LIN {X 0,Y 238.062,Z 428.573,A -85,B 0,C 180,E1 -19850.136,E2 -19850.136} C_VEL
LIN {X 0,Y 238.193,Z 430.072,A -85,B 0,C 180,E1 -19851.55,E2 -19851.55} C_VEL
LIN {X 0,Y 238.018,Z 431.292,A -85,B 0,C 180,E1 -19852.418,E2 -19852.418} C_VEL
LIN {X 0,Y 236.97,Z 433.958,A -85,B 0,C 180,E1 -19853.62,E2 -19853.62} C_VEL
LIN {X 0,Y 235.097,Z 438.66,A -85,B 0,C 180,E1 -19855.04,E2 -19855.04} C_VEL
LIN {X 0,Y 233.913,Z 444.412,A -85,B 0,C 180,E1 -19856.262,E2 -19856.262} C_VEL
LIN {X 0,Y 234.035,Z 447.586,A -85,B 0,C 180,E1 -19856.783,E2 -19856.783} C_VEL
LIN {X 0,Y 234.365,Z 449.217,A -85,B 0,C 180,E1 -19857.013,E2 -19857.013} C_VEL
LIN {X 0,Y 236.886,Z 461.103,A -85,B 0,C 180,E1 -19858.596,E2 -19858.596} C_VEL
LIN {X 0,Y 238.32,Z 473.094,A -85,B 0,C 180,E1 -19860.33,E2 -19860.33} C_VEL
LIN {X 0,Y 238.753,Z 483.531,A -85,B 0,C 180,E1 -19862.018,E2 -19862.018} C_VEL
LIN {X 0,Y 238.228,Z 494.327,A -85,B 0,C 180,E1 -19863.975,E2 -19863.975} C_VEL
LIN {X 0,Y 237.637,Z 499.757,A -85,B 0,C 180,E1 -19865.079,E2 -19865.079} C_VEL
LIN {X 0,Y 234.929,Z 509.023,A -85,B 0,C 180,E1 -19867.118,E2 -19867.118} C_VEL
LIN {X 0,Y 232.462,Z 517.532,A -85,B 0,C 180,E1 -19869.477,E2 -19869.477} C_VEL
LIN {X 0,Y 230.541,Z 524.271,A -85,B 0,C 180,E1 -19871.796,E2 -19871.796} C_VEL
LIN {X 0,Y 228.448,Z 531.313,A -85,B 0,C 180,E1 -19874.845,E2 -19874.845} C_VEL
LIN {X 0,Y 227.148,Z 536.006,A -85,B 0,C 180,E1 -19877.495,E2 -19877.495} C_VEL
LIN {X 0,Y 226.352,Z 539.618,A -85,B 0,C 180,E1 -19880.171,E2 -19880.171} C_VEL
LIN {X 0,Y 225.933,Z 542.238,A -85,B 0,C 180,E1 -19882.856,E2 -19882.856} C_VEL
LIN {X 0,Y 225.84,Z 543.543,A -85,B 0,C 180,E1 -19884.763,E2 -19884.763} C_VEL
LIN {X 0,Y 225.889,Z 544.696,A -85,B 0,C 180,E1 -19888.221,E2 -19888.221} C_VEL
LIN {X 0,Y 225.953,Z 544.713,A -85,B 0,C 180,E1 -19890.003,E2 -19890.003} C_VEL
LIN {X 0,Y 225.91,Z 544.321,A -85,B 0,C 180,E1 -19891.786,E2 -19891.786} C_VEL
LIN {X 0,Y 225.867,Z 543.479,A -85,B 0,C 180,E1 -19893.571,E2 -19893.571} C_VEL
LIN {X 0,Y 225.885,Z 542.225,A -85,B 0,C 180,E1 -19895.359,E2 -19895.359} C_VEL
LIN {X 0,Y 226.081,Z 539.542,A -85,B 0,C 180,E1 -19898.045,E2 -19898.045} C_VEL
LIN {X 0,Y 226.599,Z 535.822,A -85,B 0,C 180,E1 -19900.728,E2 -19900.728} C_VEL
LIN {X 0,Y 227.467,Z 530.966,A -85,B 0,C 180,E1 -19903.402,E2 -19903.402} C_VEL
LIN {X 0,Y 228.942,Z 524.853,A -85,B 0,C 180,E1 -19906.041,E2 -19906.041} C_VEL
LIN {X 0,Y 230.743,Z 517.238,A -85,B 0,C 180,E1 -19908.655,E2 -19908.655} C_VEL
LIN {X 0,Y 232.402,Z 509.436,A -85,B 0,C 180,E1 -19910.816,E2 -19910.816} C_VEL
LIN {X 0,Y 234.829,Z 498.867,A -85,B 0,C 180,E1 -19913.132,E2 -19913.132} C_VEL
LIN {X 0,Y 235.617,Z 494.346,A -85,B 0,C 180,E1 -19913.982,E2 -19913.982} C_VEL
LIN {X 0,Y 235.579,Z 482.776,A -85,B 0,C 180,E1 -19915.998,E2 -19915.998} C_VEL
LIN {X 0,Y 234.967,Z 472.552,A -85,B 0,C 180,E1 -19917.491,E2 -19917.491} C_VEL
LIN {X 0,Y 233.612,Z 460.76,A -85,B 0,C 180,E1 -19918.948,E2 -19918.948} C_VEL
LIN {X 0,Y 231.304,Z 447.577,A -85,B 0,C 180,E1 -19920.3,E2 -19920.3} C_VEL
LIN {X 0,Y 229.088,Z 437.272,A -85,B 0,C 180,E1 -19921.202,E2 -19921.202} C_VEL
LIN {X 0,Y 230.382,Z 432.178,A -85,B 0,C 180,E1 -19925.426,E2 -19925.426} C_VEL
LIN {X 0,Y 230.808,Z 429.565,A -85,B 0,C 180,E1 -19927.656,E2 -19927.656} C_VEL
LIN {X 0,Y 230.517,Z 426.609,A -85,B 0,C 180,E1 -19930.341,E2 -19930.341} C_VEL
LIN {X 0,Y 230.09,Z 423.947,A -85,B 0,C 180,E1 -19932.855,E2 -19932.855} C_VEL
LIN {X 0,Y 229.167,Z 419.29,A -85,B 0,C 180,E1 -19937.57,E2 -19937.57} C_VEL
LIN {X 0,Y 228.448,Z 415.194,A -85,B 0,C 180,E1 -19942.027,E2 -19942.027} C_VEL
LIN {X 0,Y 227.929,Z 412.095,A -85,B 0,C 180,E1 -19945.755,E2 -19945.755} C_VEL
LIN {X 0,Y 227.913,Z 412.099,A -85,B 0,C 180,E1 -19950.437,E2 -19950.437} C_VEL
LIN {X 0,Y 227.938,Z 412.094,A -85,B 0,C 180,E1 -19954.427,E2 -19954.427} C_VEL
LIN {X 0,Y 227.972,Z 412.09,A -85,B 0,C 180,E1 -19958.288,E2 -19958.288} C_VEL
LIN {X 0,Y 228.044,Z 412.083,A -85,B 0,C 180,E1 -19962.826,E2 -19962.826} C_VEL
LIN {X 0,Y 228.081,Z 412.077,A -85,B 0,C 180,E1 -19967.543,E2 -19967.543} C_VEL
LIN {X 0,Y 228.277,Z 412.051,A -85,B 0,C 180,E1 -19971.145,E2 -19971.145} C_VEL
LIN {X 0,Y 228.332,Z 412.044,A -85,B 0,C 180,E1 -19972.928,E2 -19972.928} C_VEL
LIN {X 0,Y 228.562,Z 412.015,A -85,B 0,C 180,E1 -19978.238,E2 -19978.238} C_VEL
LIN {X 0,Y 228.562,Z 412.015,A -85,B 0,C 180,E1 -19981.762,E2 -19981.762} C_VEL
LIN {X 0,Y 228.363,Z 412.013,A -85,B 0,C 180,E1 -19987.071,E2 -19987.071} C_VEL
LIN {X 0,Y 228.173,Z 412.057,A -85,B 0,C 180,E1 -19990.65,E2 -19990.65} C_VEL
LIN {X 0,Y 228.072,Z 412.074,A -85,B 0,C 180,E1 -19994.272,E2 -19994.272} C_VEL
LIN {X 0,Y 228.012,Z 412.068,A -85,B 0,C 180,E1 -19997.952,E2 -19997.952} C_VEL
LIN {X 0,Y 227.939,Z 412.081,A -85,B 0,C 180,E1 -20002.328,E2 -20002.328} C_VEL
LIN {X 0,Y 227.951,Z 412.089,A -85,B 0,C 180,E1 -20006.601,E2 -20006.601} C_VEL
LIN {X 0,Y 227.905,Z 412.086,A -85,B 0,C 180,E1 -20010.289,E2 -20010.289} C_VEL
LIN {X 0,Y 227.885,Z 412.081,A -85,B 0,C 180,E1 -20013.719,E2 -20013.719} C_VEL
LIN {X 0,Y 227.852,Z 412.101,A -85,B 0,C 180,E1 -20018.089,E2 -20018.089} C_VEL
LIN {X 0,Y 227.82,Z 412.094,A -85,B 0,C 180,E1 -20022.74,E2 -20022.74} C_VEL
LIN {X 0,Y 227.82,Z 412.106,A -85,B 0,C 180,E1 -20027.256,E2 -20027.256} C_VEL
LIN {X 0,Y 227.85,Z 412.092,A -85,B 0,C 180,E1 -20031.907,E2 -20031.907} C_VEL
LIN {X 0,Y 227.886,Z 412.1,A -85,B 0,C 180,E1 -20036.375,E2 -20036.375} C_VEL
LIN {X 0,Y 227.925,Z 412.087,A -85,B 0,C 180,E1 -20040.435,E2 -20040.435} C_VEL
LIN {X 0,Y 227.934,Z 412.097,A -85,B 0,C 180,E1 -20044.423,E2 -20044.423} C_VEL
LIN {X 0,Y 227.968,Z 412.09,A -85,B 0,C 180,E1 -20048.284,E2 -20048.284} C_VEL
LIN {X 0,Y 228.039,Z 412.081,A -85,B 0,C 180,E1 -20052.823,E2 -20052.823} C_VEL
LIN {X 0,Y 228.001,Z 412.084,A -85,B 0,C 180,E1 -20055.721,E2 -20055.721} C_VEL
LIN {X 0,Y 227.831,Z 412.107,A -85,B 0,C 180,E1 -20059.331,E2 -20059.331} C_VEL
LIN {X 0,Y 227.966,Z 413.662,A -85,B 0,C 180,E1 -20061.911,E2 -20061.911} C_VEL
LIN {X 0,Y 228.963,Z 416.695,A -85,B 0,C 180,E1 -20062.223,E2 -20062.223} C_VEL
LIN {X 0,Y 232.416,Z 426.574,A -85,B 0,C 180,E1 -20063.349,E2 -20063.349} C_VEL
LIN {X 0,Y 235.589,Z 438.414,A -85,B 0,C 180,E1 -20064.862,E2 -20064.862} C_VEL
LIN {X 0,Y 238.196,Z 450.137,A -85,B 0,C 180,E1 -20066.614,E2 -20066.614} C_VEL
LIN {X 0,Y 239.333,Z 457.179,A -85,B 0,C 180,E1 -20067.804,E2 -20067.804} C_VEL
LIN {X 0,Y 237.285,Z 468.194,A -85,B 0,C 180,E1 -20069.572,E2 -20069.572} C_VEL
LIN {X 0,Y 235.429,Z 476.783,A -85,B 0,C 180,E1 -20071.28,E2 -20071.28} C_VEL
LIN {X 0,Y 233.317,Z 485.711,A -85,B 0,C 180,E1 -20073.45,E2 -20073.45} C_VEL
LIN {X 0,Y 231.223,Z 494.31,A -85,B 0,C 180,E1 -20076.103,E2 -20076.103} C_VEL
LIN {X 0,Y 229.481,Z 501.232,A -85,B 0,C 180,E1 -20078.805,E2 -20078.805} C_VEL
LIN {X 0,Y 228.149,Z 506.729,A -85,B 0,C 180,E1 -20081.547,E2 -20081.547} C_VEL
LIN {X 0,Y 227.164,Z 510.978,A -85,B 0,C 180,E1 -20084.326,E2 -20084.326} C_VEL
LIN {X 0,Y 226.609,Z 513.168,A -85,B 0,C 180,E1 -20086.204,E2 -20086.204} C_VEL
LIN {X 0,Y 226.171,Z 514.914,A -85,B 0,C 180,E1 -20088.1,E2 -20088.1} C_VEL
LIN {X 0,Y 225.826,Z 516.659,A -85,B 0,C 180,E1 -20090.99,E2 -20090.99} C_VEL
LIN {X 0,Y 225.784,Z 517.355,A -85,B 0,C 180,E1 -20093.865,E2 -20093.865} C_VEL
LIN {X 0,Y 225.956,Z 517.249,A -85,B 0,C 180,E1 -20095.809,E2 -20095.809} C_VEL
LIN {X 0,Y 226.278,Z 516.652,A -85,B 0,C 180,E1 -20097.763,E2 -20097.763} C_VEL
LIN {X 0,Y 226.766,Z 515.562,A -85,B 0,C 180,E1 -20099.798,E2 -20099.798} C_VEL
LIN {X 0,Y 227.73,Z 513.054,A -85,B 0,C 180,E1 -20102.684,E2 -20102.684} C_VEL
LIN {X 0,Y 229.073,Z 509.227,A -85,B 0,C 180,E1 -20105.651,E2 -20105.651} C_VEL
LIN {X 0,Y 230.932,Z 504.002,A -85,B 0,C 180,E1 -20108.595,E2 -20108.595} C_VEL
LIN {X 0,Y 233.221,Z 497.184,A -85,B 0,C 180,E1 -20111.52,E2 -20111.52} C_VEL
LIN {X 0,Y 235.505,Z 490.026,A -85,B 0,C 180,E1 -20113.908,E2 -20113.908} C_VEL
LIN {X 0,Y 238.122,Z 480.988,A -85,B 0,C 180,E1 -20116.305,E2 -20116.305} C_VEL
LIN {X 0,Y 240.681,Z 471.659,A -85,B 0,C 180,E1 -20118.265,E2 -20118.265} C_VEL
LIN {X 0,Y 242.859,Z 462.006,A -85,B 0,C 180,E1 -20119.918,E2 -20119.918} C_VEL
LIN {X 0,Y 241.384,Z 452.108,A -85,B 0,C 180,E1 -20121.817,E2 -20121.817} C_VEL
LIN {X 0,Y 238.809,Z 441.764,A -85,B 0,C 180,E1 -20123.682,E2 -20123.682} C_VEL
LIN {X 0,Y 234.757,Z 430.297,A -85,B 0,C 180,E1 -20125.658,E2 -20125.658} C_VEL
LIN {X 0,Y 230.034,Z 420.138,A -85,B 0,C 180,E1 -20127.42,E2 -20127.42} C_VEL
LIN {X 0,Y 228.43,Z 417.231,A -85,B 0,C 180,E1 -20127.946,E2 -20127.946} C_VEL
LIN {X 0,Y 228.162,Z 416.054,A -85,B 0,C 180,E1 -20128.164,E2 -20128.164} C_VEL
LIN {X 0,Y 228.225,Z 414.903,A -85,B 0,C 180,E1 -20130.481,E2 -20130.481} C_VEL
LIN {X 0,Y 228.082,Z 413.1,A -85,B 0,C 180,E1 -20134.444,E2 -20134.444} C_VEL
LIN {X 0,Y 227.967,Z 412.089,A -85,B 0,C 180,E1 -20137.637,E2 -20137.637} C_VEL
LIN {X 0,Y 228.029,Z 412.081,A -85,B 0,C 180,E1 -20142.816,E2 -20142.816} C_VEL
LIN {X 0,Y 228.057,Z 412.074,A -85,B 0,C 180,E1 -20147.542,E2 -20147.542} C_VEL
LIN {X 0,Y 228.289,Z 412.049,A -85,B 0,C 180,E1 -20151.146,E2 -20151.146} C_VEL
LIN {X 0,Y 228.339,Z 412.036,A -85,B 0,C 180,E1 -20152.928,E2 -20152.928} C_VEL
LIN {X 0,Y 228.539,Z 412.018,A -85,B 0,C 180,E1 -20158.238,E2 -20158.238} C_VEL
LIN {X 0,Y 228.548,Z 412.017,A -85,B 0,C 180,E1 -20161.762,E2 -20161.762} C_VEL
LIN {X 0,Y 228.338,Z 412.042,A -85,B 0,C 180,E1 -20167.072,E2 -20167.072} C_VEL
LIN {X 0,Y 228.147,Z 412.065,A -85,B 0,C 180,E1 -20170.651,E2 -20170.651} C_VEL
LIN {X 0,Y 228.049,Z 412.079,A -85,B 0,C 180,E1 -20176.103,E2 -20176.103} C_VEL
LIN {X 0,Y 227.956,Z 412.093,A -85,B 0,C 180,E1 -20179.824,E2 -20179.824} C_VEL
LIN {X 0,Y 227.926,Z 412.098,A -85,B 0,C 180,E1 -20183.631,E2 -20183.631} C_VEL
LIN {X 0,Y 227.927,Z 412.179,A -85,B 0,C 180,E1 -20186.604,E2 -20186.604} C_VEL
LIN {X 0,Y 228.294,Z 414.25,A -85,B 0,C 180,E1 -20190.47,E2 -20190.47} C_VEL
LIN {X 0,Y 228.65,Z 416.385,A -85,B 0,C 180,E1 -20193.92,E2 -20193.92} C_VEL
LIN {X 0,Y 229.122,Z 419.126,A -85,B 0,C 180,E1 -20197.841,E2 -20197.841} C_VEL
LIN {X 0,Y 229.772,Z 422.616,A -85,B 0,C 180,E1 -20202.292,E2 -20202.292} C_VEL
LIN {X 0,Y 230.273,Z 425.329,A -85,B 0,C 180,E1 -20205.421,E2 -20205.421} C_VEL
LIN {X 0,Y 231.075,Z 429.962,A -85,B 0,C 180,E1 -20210.31,E2 -20210.31} C_VEL
LIN {X 0,Y 231.136,Z 432.295,A -85,B 0,C 180,E1 -20212.551,E2 -20212.551} C_VEL
LIN {X 0,Y 230.382,Z 435.405,A -85,B 0,C 180,E1 -20215.31,E2 -20215.31} C_VEL
LIN {X 0,Y 231.399,Z 439.104,A -85,B 0,C 180,E1 -20215.736,E2 -20215.736} C_VEL
LIN {X 0,Y 234.365,Z 449.217,A -85,B 0,C 180,E1 -20217.013,E2 -20217.013} C_VEL
LIN {X 0,Y 235.145,Z 454.521,A -85,B 0,C 180,E1 -20217.622,E2 -20217.622} C_VEL
LIN {X 0,Y 234.907,Z 460.061,A -85,B 0,C 180,E1 -20218.15,E2 -20218.15} C_VEL
LIN {X 0,Y 232.877,Z 471.151,A -85,B 0,C 180,E1 -20219.213,E2 -20219.213} C_VEL
LIN {X 0,Y 232.213,Z 476.411,A -85,B 0,C 180,E1 -20219.895,E2 -20219.895} C_VEL
LIN {X 0,Y 232.214,Z 478.052,A -85,B 0,C 180,E1 -20220.162,E2 -20220.162} C_VEL
LIN {X 0,Y 232.218,Z 487.546,A -85,B 0,C 180,E1 -20221.842,E2 -20221.842} C_VEL
LIN {X 0,Y 231.311,Z 498.773,A -85,B 0,C 180,E1 -20224.107,E2 -20224.107} C_VEL
LIN {X 0,Y 228.933,Z 507.277,A -85,B 0,C 180,E1 -20226.003,E2 -20226.003} C_VEL
LIN {X 0,Y 226.464,Z 515.184,A -85,B 0,C 180,E1 -20228.14,E2 -20228.14} C_VEL
LIN {X 0,Y 224.608,Z 521.778,A -85,B 0,C 180,E1 -20230.348,E2 -20230.348} C_VEL
LIN {X 0,Y 222.759,Z 527.294,A -85,B 0,C 180,E1 -20232.563,E2 -20232.563} C_VEL
LIN {X 0,Y 221.019,Z 532.729,A -85,B 0,C 180,E1 -20235.267,E2 -20235.267} C_VEL
LIN {X 0,Y 219.857,Z 537.009,A -85,B 0,C 180,E1 -20238.012,E2 -20238.012} C_VEL
LIN {X 0,Y 219.14,Z 540.246,A -85,B 0,C 180,E1 -20240.776,E2 -20240.776} C_VEL
LIN {X 0,Y 218.857,Z 541.881,A -85,B 0,C 180,E1 -20242.624,E2 -20242.624} C_VEL
LIN {X 0,Y 218.741,Z 543.288,A -85,B 0,C 180,E1 -20244.884,E2 -20244.884} C_VEL
LIN {X 0,Y 218.819,Z 544.273,A -85,B 0,C 180,E1 -20248.163,E2 -20248.163} C_VEL
LIN {X 0,Y 218.881,Z 544.273,A -85,B 0,C 180,E1 -20250.004,E2 -20250.004} C_VEL
LIN {X 0,Y 218.839,Z 543.855,A -85,B 0,C 180,E1 -20251.844,E2 -20251.844} C_VEL
LIN {X 0,Y 218.787,Z 541.941,A -85,B 0,C 180,E1 -20255.25,E2 -20255.25} C_VEL
LIN {X 0,Y 219.044,Z 539.001,A -85,B 0,C 180,E1 -20258.305,E2 -20258.305} C_VEL
LIN {X 0,Y 219.601,Z 535.242,A -85,B 0,C 180,E1 -20261.074,E2 -20261.074} C_VEL
LIN {X 0,Y 220.535,Z 530.346,A -85,B 0,C 180,E1 -20263.831,E2 -20263.831} C_VEL
LIN {X 0,Y 222.039,Z 524.181,A -85,B 0,C 180,E1 -20266.554,E2 -20266.554} C_VEL
LIN {X 0,Y 223.872,Z 516.817,A -85,B 0,C 180,E1 -20269.143,E2 -20269.143} C_VEL
LIN {X 0,Y 225.74,Z 508.627,A -85,B 0,C 180,E1 -20271.461,E2 -20271.461} C_VEL
LIN {X 0,Y 228.022,Z 499.037,A -85,B 0,C 180,E1 -20273.624,E2 -20273.624} C_VEL
LIN {X 0,Y 228.734,Z 495.768,A -85,B 0,C 180,E1 -20274.268,E2 -20274.268} C_VEL
LIN {X 0,Y 228.819,Z 484.478,A -85,B 0,C 180,E1 -20276.349,E2 -20276.349} C_VEL
LIN {X 0,Y 228.246,Z 473.362,A -85,B 0,C 180,E1 -20278.075,E2 -20278.075} C_VEL
LIN {X 0,Y 227.048,Z 462.033,A -85,B 0,C 180,E1 -20279.565,E2 -20279.565} C_VEL
LIN {X 0,Y 224.921,Z 449.232,A -85,B 0,C 180,E1 -20280.979,E2 -20280.979} C_VEL
LIN {X 0,Y 222.238,Z 436.912,A -85,B 0,C 180,E1 -20282.094,E2 -20282.094} C_VEL
LIN {X 0,Y 223.586,Z 431.582,A -85,B 0,C 180,E1 -20286.675,E2 -20286.675} C_VEL
LIN {X 0,Y 223.692,Z 429.1,A -85,B 0,C 180,E1 -20288.933,E2 -20288.933} C_VEL
LIN {X 0,Y 222.94,Z 424.38,A -85,B 0,C 180,E1 -20293.526,E2 -20293.526} C_VEL
LIN {X 0,Y 222.368,Z 421.37,A -85,B 0,C 180,E1 -20296.633,E2 -20296.633} C_VEL
LIN {X 0,Y 221.66,Z 417.726,A -85,B 0,C 180,E1 -20300.645,E2 -20300.645} C_VEL
LIN {X 0,Y 221.385,Z 415.755,A -85,B 0,C 180,E1 -20302.903,E2 -20302.903} C_VEL
LIN {X 0,Y 220.851,Z 412.978,A -85,B 0,C 180,E1 -20306.518,E2 -20306.518} C_VEL
LIN {X 0,Y 220.843,Z 412.979,A -85,B 0,C 180,E1 -20309.391,E2 -20309.391} C_VEL
LIN {X 0,Y 220.904,Z 412.967,A -85,B 0,C 180,E1 -20313.55,E2 -20313.55} C_VEL
LIN {X 0,Y 220.887,Z 412.97,A -85,B 0,C 180,E1 -20317.554,E2 -20317.554} C_VEL
LIN {X 0,Y 220.994,Z 412.963,A -85,B 0,C 180,E1 -20322.572,E2 -20322.572} C_VEL
LIN {X 0,Y 221.02,Z 412.957,A -85,B 0,C 180,E1 -20327.139,E2 -20327.139} C_VEL
LIN {X 0,Y 221.214,Z 412.932,A -85,B 0,C 180,E1 -20330.86,E2 -20330.86} C_VEL
LIN {X 0,Y 221.268,Z 412.925,A -85,B 0,C 180,E1 -20332.701,E2 -20332.701} C_VEL
LIN {X 0,Y 221.52,Z 412.893,A -85,B 0,C 180,E1 -20338.182,E2 -20338.182} C_VEL
LIN {X 0,Y 221.52,Z 412.892,A -85,B 0,C 180,E1 -20341.818,E2 -20341.818} C_VEL
LIN {X 0,Y 221.299,Z 412.892,A -85,B 0,C 180,E1 -20347.298,E2 -20347.298} C_VEL
LIN {X 0,Y 221.121,Z 412.935,A -85,B 0,C 180,E1 -20350.994,E2 -20350.994} C_VEL
LIN {X 0,Y 221.025,Z 412.945,A -85,B 0,C 180,E1 -20356.629,E2 -20356.629} C_VEL
LIN {X 0,Y 220.901,Z 412.944,A -85,B 0,C 180,E1 -20360.485,E2 -20360.485} C_VEL
LIN {X 0,Y 220.876,Z 412.968,A -85,B 0,C 180,E1 -20364.434,E2 -20364.434} C_VEL
LIN {X 0,Y 220.836,Z 412.973,A -85,B 0,C 180,E1 -20368.514,E2 -20368.514} C_VEL
LIN {X 0,Y 220.825,Z 412.955,A -85,B 0,C 180,E1 -20372.755,E2 -20372.755} C_VEL
LIN {X 0,Y 220.818,Z 412.978,A -85,B 0,C 180,E1 -20377.277,E2 -20377.277} C_VEL
LIN {X 0,Y 220.778,Z 412.973,A -85,B 0,C 180,E1 -20381.951,E2 -20381.951} C_VEL
LIN {X 0,Y 220.783,Z 412.975,A -85,B 0,C 180,E1 -20385.545,E2 -20385.545} C_VEL
LIN {X 0,Y 220.814,Z 412.977,A -85,B 0,C 180,E1 -20390.461,E2 -20390.461} C_VEL
LIN {X 0,Y 220.808,Z 412.98,A -85,B 0,C 180,E1 -20395.043,E2 -20395.043} C_VEL
LIN {X 0,Y 220.875,Z 412.965,A -85,B 0,C 180,E1 -20399.393,E2 -20399.393} C_VEL
LIN {X 0,Y 220.901,Z 412.972,A -85,B 0,C 180,E1 -20403.547,E2 -20403.547} C_VEL
LIN {X 0,Y 220.884,Z 412.972,A -85,B 0,C 180,E1 -20407.551,E2 -20407.551} C_VEL
LIN {X 0,Y 220.989,Z 412.958,A -85,B 0,C 180,E1 -20412.568,E2 -20412.568} C_VEL
LIN {X 0,Y 220.902,Z 412.97,A -85,B 0,C 180,E1 -20417.129,E2 -20417.129} C_VEL
LIN {X 0,Y 220.798,Z 412.983,A -85,B 0,C 180,E1 -20418.987,E2 -20418.987} C_VEL
LIN {X 0,Y 220.954,Z 414.219,A -85,B 0,C 180,E1 -20420.969,E2 -20420.969} C_VEL
LIN {X 0,Y 223.204,Z 420.164,A -85,B 0,C 180,E1 -20421.643,E2 -20421.643} C_VEL
LIN {X 0,Y 226.361,Z 429.527,A -85,B 0,C 180,E1 -20422.807,E2 -20422.807} C_VEL
LIN {X 0,Y 229.489,Z 441.911,A -85,B 0,C 180,E1 -20424.505,E2 -20424.505} C_VEL
LIN {X 0,Y 232.066,Z 454.263,A -85,B 0,C 180,E1 -20426.524,E2 -20426.524} C_VEL
LIN {X 0,Y 232.632,Z 458.252,A -85,B 0,C 180,E1 -20427.238,E2 -20427.238} C_VEL
LIN {X 0,Y 230.456,Z 469.524,A -85,B 0,C 180,E1 -20429.123,E2 -20429.123} C_VEL
LIN {X 0,Y 228.084,Z 479.834,A -85,B 0,C 180,E1 -20431.321,E2 -20431.321} C_VEL
LIN {X 0,Y 226.029,Z 488.247,A -85,B 0,C 180,E1 -20433.562,E2 -20433.562} C_VEL
LIN {X 0,Y 223.916,Z 496.488,A -85,B 0,C 180,E1 -20436.303,E2 -20436.303} C_VEL
LIN {X 0,Y 222.197,Z 503.03,A -85,B 0,C 180,E1 -20439.096,E2 -20439.096} C_VEL
LIN {X 0,Y 220.896,Z 508.209,A -85,B 0,C 180,E1 -20441.931,E2 -20441.931} C_VEL
LIN {X 0,Y 219.911,Z 512.199,A -85,B 0,C 180,E1 -20444.809,E2 -20444.809} C_VEL
LIN {X 0,Y 219.362,Z 514.271,A -85,B 0,C 180,E1 -20446.755,E2 -20446.755} C_VEL
LIN {X 0,Y 218.986,Z 515.837,A -85,B 0,C 180,E1 -20448.715,E2 -20448.715} C_VEL
LIN {X 0,Y 218.716,Z 517.207,A -85,B 0,C 180,E1 -20451.274,E2 -20451.274} C_VEL
LIN {X 0,Y 218.752,Z 517.802,A -85,B 0,C 180,E1 -20454.682,E2 -20454.682} C_VEL
LIN {X 0,Y 218.984,Z 517.527,A -85,B 0,C 180,E1 -20456.695,E2 -20456.695} C_VEL
LIN {X 0,Y 219.387,Z 516.804,A -85,B 0,C 180,E1 -20458.715,E2 -20458.715} C_VEL
LIN {X 0,Y 219.957,Z 515.542,A -85,B 0,C 180,E1 -20460.741,E2 -20460.741} C_VEL
LIN {X 0,Y 220.658,Z 513.801,A -85,B 0,C 180,E1 -20462.778,E2 -20462.778} C_VEL
LIN {X 0,Y 222.074,Z 510.148,A -85,B 0,C 180,E1 -20465.831,E2 -20465.831} C_VEL
LIN {X 0,Y 223.982,Z 505.078,A -85,B 0,C 180,E1 -20468.864,E2 -20468.864} C_VEL
LIN {X 0,Y 226.297,Z 498.577,A -85,B 0,C 180,E1 -20471.81,E2 -20471.81} C_VEL
LIN {X 0,Y 228.727,Z 491.424,A -85,B 0,C 180,E1 -20474.343,E2 -20474.343} C_VEL
LIN {X 0,Y 231.418,Z 482.709,A -85,B 0,C 180,E1 -20476.785,E2 -20476.785} C_VEL
LIN {X 0,Y 234.248,Z 473.007,A -85,B 0,C 180,E1 -20478.915,E2 -20478.915} C_VEL
LIN {X 0,Y 236.481,Z 463.65,A -85,B 0,C 180,E1 -20480.59,E2 -20480.59} C_VEL
LIN {X 0,Y 235.193,Z 454.325,A -85,B 0,C 180,E1 -20482.494,E2 -20482.494} C_VEL
LIN {X 0,Y 232.854,Z 444.498,A -85,B 0,C 180,E1 -20484.389,E2 -20484.389} C_VEL
LIN {X 0,Y 229.068,Z 433.296,A -85,B 0,C 180,E1 -20486.478,E2 -20486.478} C_VEL
LIN {X 0,Y 225.11,Z 424.544,A -85,B 0,C 180,E1 -20488.125,E2 -20488.125} C_VEL
LIN {X 0,Y 222.759,Z 420.245,A -85,B 0,C 180,E1 -20488.974,E2 -20488.974} C_VEL
LIN {X 0,Y 221.424,Z 417.451,A -85,B 0,C 180,E1 -20489.48,E2 -20489.48} C_VEL
LIN {X 0,Y 221.238,Z 416.651,A -85,B 0,C 180,E1 -20489.584,E2 -20489.584} C_VEL
LIN {X 0,Y 221.15,Z 414.855,A -85,B 0,C 180,E1 -20493.582,E2 -20493.582} C_VEL
LIN {X 0,Y 220.974,Z 413.261,A -85,B 0,C 180,E1 -20497.564,E2 -20497.564} C_VEL
LIN {X 0,Y 220.919,Z 412.965,A -85,B 0,C 180,E1 -20501.451,E2 -20501.451} C_VEL
LIN {X 0,Y 220.98,Z 412.959,A -85,B 0,C 180,E1 -20505.26,E2 -20505.26} C_VEL
LIN {X 0,Y 221.22,Z 412.927,A -85,B 0,C 180,E1 -20510.86,E2 -20510.86} C_VEL
LIN {X 0,Y 221.274,Z 412.916,A -85,B 0,C 180,E1 -20512.701,E2 -20512.701} C_VEL
LIN {X 0,Y 221.497,Z 412.895,A -85,B 0,C 180,E1 -20518.182,E2 -20518.182} C_VEL
LIN {X 0,Y 221.507,Z 412.894,A -85,B 0,C 180,E1 -20521.818,E2 -20521.818} C_VEL
LIN {X 0,Y 221.273,Z 412.922,A -85,B 0,C 180,E1 -20527.299,E2 -20527.299} C_VEL
LIN {X 0,Y 221.096,Z 412.944,A -85,B 0,C 180,E1 -20530.995,E2 -20530.995} C_VEL
LIN {X 0,Y 221.009,Z 412.957,A -85,B 0,C 180,E1 -20536.631,E2 -20536.631} C_VEL
LIN {X 0,Y 220.911,Z 412.969,A -85,B 0,C 180,E1 -20540.485,E2 -20540.485} C_VEL
LIN {X 0,Y 220.868,Z 412.978,A -85,B 0,C 180,E1 -20544.435,E2 -20544.435} C_VEL
LIN {X 0,Y 221.153,Z 414.834,A -85,B 0,C 180,E1 -20548.469,E2 -20548.469} C_VEL
LIN {X 0,Y 221.57,Z 417.191,A -85,B 0,C 180,E1 -20552.631,E2 -20552.631} C_VEL
LIN {X 0,Y 222.1,Z 420.025,A -85,B 0,C 180,E1 -20556.958,E2 -20556.958} C_VEL
LIN {X 0,Y 222.675,Z 423.425,A -85,B 0,C 180,E1 -20561.514,E2 -20561.514} C_VEL
LIN {X 0,Y 223.444,Z 427.477,A -85,B 0,C 180,E1 -20566.338,E2 -20566.338} C_VEL
LIN {X 0,Y 224.06,Z 430.924,A -85,B 0,C 180,E1 -20570.058,E2 -20570.058} C_VEL
LIN {X 0,Y 224.121,Z 432.479,A -85,B 0,C 180,E1 -20571.624,E2 -20571.624} C_VEL
LIN {X 0,Y 223.761,Z 435.016,A -85,B 0,C 180,E1 -20573.943,E2 -20573.943} C_VEL
LIN {X 0,Y 224.665,Z 438.369,A -85,B 0,C 180,E1 -20574.332,E2 -20574.332} C_VEL
LIN {X 0,Y 227.684,Z 448.099,A -85,B 0,C 180,E1 -20575.665,E2 -20575.665} C_VEL
LIN {X 0,Y 230.286,Z 459.729,A -85,B 0,C 180,E1 -20577.317,E2 -20577.317} C_VEL
LIN {X 0,Y 231.744,Z 470.737,A -85,B 0,C 180,E1 -20578.97,E2 -20578.97} C_VEL
LIN {X 0,Y 232.214,Z 478.052,A -85,B 0,C 180,E1 -20580.162,E2 -20580.162} C_VEL
LIN {X 0,Y 231.785,Z 483.089,A -85,B 0,C 180,E1 -20580.95,E2 -20580.95} C_VEL
LIN {X 0,Y 230.348,Z 488.088,A -85,B 0,C 180,E1 -20581.679,E2 -20581.679} C_VEL
LIN {X 0,Y 226.133,Z 497.627,A -85,B 0,C 180,E1 -20583.173,E2 -20583.173} C_VEL
LIN {X 0,Y 223.687,Z 503.561,A -85,B 0,C 180,E1 -20584.359,E2 -20584.359} C_VEL
LIN {X 0,Y 220.85,Z 512.145,A -85,B 0,C 180,E1 -20586.565,E2 -20586.565} C_VEL
LIN {X 0,Y 218.171,Z 520.4,A -85,B 0,C 180,E1 -20589.251,E2 -20589.251} C_VEL
LIN {X 0,Y 216.268,Z 526.073,A -85,B 0,C 180,E1 -20591.532,E2 -20591.532} C_VEL
LIN {X 0,Y 214.14,Z 532.48,A -85,B 0,C 180,E1 -20594.782,E2 -20594.782} C_VEL
LIN {X 0,Y 212.872,Z 536.716,A -85,B 0,C 180,E1 -20597.612,E2 -20597.612} C_VEL
LIN {X 0,Y 212.099,Z 539.913,A -85,B 0,C 180,E1 -20600.467,E2 -20600.467} C_VEL
LIN {X 0,Y 211.81,Z 541.53,A -85,B 0,C 180,E1 -20602.377,E2 -20602.377} C_VEL
LIN {X 0,Y 211.643,Z 543.035,A -85,B 0,C 180,E1 -20605.01,E2 -20605.01} C_VEL
LIN {X 0,Y 211.749,Z 543.849,A -85,B 0,C 180,E1 -20608.102,E2 -20608.102} C_VEL
LIN {X 0,Y 211.81,Z 543.831,A -85,B 0,C 180,E1 -20610.004,E2 -20610.004} C_VEL
LIN {X 0,Y 211.77,Z 543.378,A -85,B 0,C 180,E1 -20611.905,E2 -20611.905} C_VEL
LIN {X 0,Y 211.723,Z 541.573,A -85,B 0,C 180,E1 -20615.23,E2 -20615.23} C_VEL
LIN {X 0,Y 211.982,Z 538.44,A -85,B 0,C 180,E1 -20618.584,E2 -20618.584} C_VEL
LIN {X 0,Y 212.597,Z 534.638,A -85,B 0,C 180,E1 -20621.444,E2 -20621.444} C_VEL
LIN {X 0,Y 213.626,Z 529.696,A -85,B 0,C 180,E1 -20624.288,E2 -20624.288} C_VEL
LIN {X 0,Y 215.161,Z 523.474,A -85,B 0,C 180,E1 -20627.099,E2 -20627.099} C_VEL
LIN {X 0,Y 217.02,Z 516.374,A -85,B 0,C 180,E1 -20629.657,E2 -20629.657} C_VEL
LIN {X 0,Y 219.089,Z 507.761,A -85,B 0,C 180,E1 -20632.146,E2 -20632.146} C_VEL
LIN {X 0,Y 221.536,Z 498.094,A -85,B 0,C 180,E1 -20634.36,E2 -20634.36} C_VEL
LIN {X 0,Y 221.989,Z 492.296,A -85,B 0,C 180,E1 -20635.557,E2 -20635.557} C_VEL
LIN {X 0,Y 221.993,Z 481.249,A -85,B 0,C 180,E1 -20637.57,E2 -20637.57} C_VEL
LIN {X 0,Y 221.139,Z 468.796,A -85,B 0,C 180,E1 -20639.467,E2 -20639.467} C_VEL
LIN {X 0,Y 219.584,Z 456.823,A -85,B 0,C 180,E1 -20641.004,E2 -20641.004} C_VEL
LIN {X 0,Y 217.129,Z 443.997,A -85,B 0,C 180,E1 -20642.386,E2 -20642.386} C_VEL
LIN {X 0,Y 215.438,Z 436.465,A -85,B 0,C 180,E1 -20643.081,E2 -20643.081} C_VEL
LIN {X 0,Y 216.563,Z 432.187,A -85,B 0,C 180,E1 -20646.9,E2 -20646.9} C_VEL
LIN {X 0,Y 216.681,Z 430.082,A -85,B 0,C 180,E1 -20648.882,E2 -20648.882} C_VEL
LIN {X 0,Y 216.013,Z 425.863,A -85,B 0,C 180,E1 -20653.101,E2 -20653.101} C_VEL
LIN {X 0,Y 215.342,Z 422.464,A -85,B 0,C 180,E1 -20656.735,E2 -20656.735} C_VEL
LIN {X 0,Y 214.508,Z 417.987,A -85,B 0,C 180,E1 -20661.847,E2 -20661.847} C_VEL
LIN {X 0,Y 213.871,Z 414.156,A -85,B 0,C 180,E1 -20666.604,E2 -20666.604} C_VEL
LIN {X 0,Y 213.784,Z 413.859,A -85,B 0,C 180,E1 -20667.151,E2 -20667.151} C_VEL
LIN {X 0,Y 213.836,Z 413.85,A -85,B 0,C 180,E1 -20672.604,E2 -20672.604} C_VEL
LIN {X 0,Y 213.862,Z 413.846,A -85,B 0,C 180,E1 -20676.954,E2 -20676.954} C_VEL
LIN {X 0,Y 213.953,Z 413.839,A -85,B 0,C 180,E1 -20682.804,E2 -20682.804} C_VEL
LIN {X 0,Y 213.961,Z 413.838,A -85,B 0,C 180,E1 -20686.707,E2 -20686.707} C_VEL
LIN {X 0,Y 214.152,Z 413.813,A -85,B 0,C 180,E1 -20690.555,E2 -20690.555} C_VEL
LIN {X 0,Y 214.107,Z 413.817,A -85,B 0,C 180,E1 -20694.349,E2 -20694.349} C_VEL
LIN {X 0,Y 214.453,Z 413.773,A -85,B 0,C 180,E1 -20698.122,E2 -20698.122} C_VEL
LIN {X 0,Y 214.555,Z 413.76,A -85,B 0,C 180,E1 -20700,E2 -20700} C_VEL
LIN {X 0,Y 214.453,Z 413.771,A -85,B 0,C 180,E1 -20701.878,E2 -20701.878} C_VEL
LIN {X 0,Y 214.237,Z 413.771,A -85,B 0,C 180,E1 -20707.54,E2 -20707.54} C_VEL
LIN {X 0,Y 214.054,Z 413.816,A -85,B 0,C 180,E1 -20711.361,E2 -20711.361} C_VEL
LIN {X 0,Y 213.942,Z 413.834,A -85,B 0,C 180,E1 -20715.236,E2 -20715.236} C_VEL
LIN {X 0,Y 213.848,Z 413.824,A -85,B 0,C 180,E1 -20719.186,E2 -20719.186} C_VEL
LIN {X 0,Y 213.857,Z 413.836,A -85,B 0,C 180,E1 -20723.226,E2 -20723.226} C_VEL
LIN {X 0,Y 213.838,Z 413.849,A -85,B 0,C 180,E1 -20727.449,E2 -20727.449} C_VEL
LIN {X 0,Y 213.776,Z 413.834,A -85,B 0,C 180,E1 -20731.736,E2 -20731.736} C_VEL
LIN {X 0,Y 213.752,Z 413.854,A -85,B 0,C 180,E1 -20736.287,E2 -20736.287} C_VEL
LIN {X 0,Y 213.72,Z 413.857,A -85,B 0,C 180,E1 -20741.123,E2 -20741.123} C_VEL
LIN {X 0,Y 213.715,Z 413.846,A -85,B 0,C 180,E1 -20743.676,E2 -20743.676} C_VEL
LIN {X 0,Y 213.715,Z 413.858,A -85,B 0,C 180,E1 -20746.342,E2 -20746.342} C_VEL
LIN {X 0,Y 213.725,Z 413.863,A -85,B 0,C 180,E1 -20749.141,E2 -20749.141} C_VEL
LIN {X 0,Y 213.75,Z 413.852,A -85,B 0,C 180,E1 -20753.709,E2 -20753.709} C_VEL
LIN {X 0,Y 213.802,Z 413.85,A -85,B 0,C 180,E1 -20758.722,E2 -20758.722} C_VEL
LIN {X 0,Y 213.832,Z 413.853,A -85,B 0,C 180,E1 -20762.601,E2 -20762.601} C_VEL
LIN {X 0,Y 213.858,Z 413.844,A -85,B 0,C 180,E1 -20766.95,E2 -20766.95} C_VEL
LIN {X 0,Y 213.948,Z 413.836,A -85,B 0,C 180,E1 -20772.801,E2 -20772.801} C_VEL
LIN {X 0,Y 213.851,Z 413.848,A -85,B 0,C 180,E1 -20776.697,E2 -20776.697} C_VEL
LIN {X 0,Y 213.755,Z 413.86,A -85,B 0,C 180,E1 -20778.619,E2 -20778.619} C_VEL
LIN {X 0,Y 213.854,Z 414.557,A -85,B 0,C 180,E1 -20779.916,E2 -20779.916} C_VEL
LIN {X 0,Y 215.01,Z 417.63,A -85,B 0,C 180,E1 -20780.289,E2 -20780.289} C_VEL
LIN {X 0,Y 219.19,Z 428.673,A -85,B 0,C 180,E1 -20781.742,E2 -20781.742} C_VEL
LIN {X 0,Y 222.194,Z 440.467,A -85,B 0,C 180,E1 -20783.387,E2 -20783.387} C_VEL
LIN {X 0,Y 224.523,Z 450.998,A -85,B 0,C 180,E1 -20785.104,E2 -20785.104} C_VEL
LIN {X 0,Y 225.945,Z 459.383,A -85,B 0,C 180,E1 -20786.649,E2 -20786.649} C_VEL
LIN {X 0,Y 223.936,Z 469.638,A -85,B 0,C 180,E1 -20788.423,E2 -20788.423} C_VEL
LIN {X 0,Y 221.687,Z 479.102,A -85,B 0,C 180,E1 -20790.451,E2 -20790.451} C_VEL
LIN {X 0,Y 219.503,Z 487.708,A -85,B 0,C 180,E1 -20792.749,E2 -20792.749} C_VEL
LIN {X 0,Y 217.259,Z 496.12,A -85,B 0,C 180,E1 -20795.565,E2 -20795.565} C_VEL
LIN {X 0,Y 215.425,Z 502.861,A -85,B 0,C 180,E1 -20798.438,E2 -20798.438} C_VEL
LIN {X 0,Y 214.032,Z 508.165,A -85,B 0,C 180,E1 -20801.359,E2 -20801.359} C_VEL
LIN {X 0,Y 212.951,Z 512.273,A -85,B 0,C 180,E1 -20804.327,E2 -20804.327} C_VEL
LIN {X 0,Y 212.131,Z 515.283,A -85,B 0,C 180,E1 -20807.344,E2 -20807.344} C_VEL
LIN {X 0,Y 211.793,Z 516.701,A -85,B 0,C 180,E1 -20809.376,E2 -20809.376} C_VEL
LIN {X 0,Y 211.612,Z 517.724,A -85,B 0,C 180,E1 -20811.576,E2 -20811.576} C_VEL
LIN {X 0,Y 211.621,Z 518.155,A -85,B 0,C 180,E1 -20813.481,E2 -20813.481} C_VEL
LIN {X 0,Y 211.861,Z 518.081,A -85,B 0,C 180,E1 -20816.406,E2 -20816.406} C_VEL
LIN {X 0,Y 212.561,Z 516.854,A -85,B 0,C 180,E1 -20819.728,E2 -20819.728} C_VEL
LIN {X 0,Y 213.218,Z 515.464,A -85,B 0,C 180,E1 -20821.824,E2 -20821.824} C_VEL
LIN {X 0,Y 214.541,Z 512.314,A -85,B 0,C 180,E1 -20825.02,E2 -20825.02} C_VEL
LIN {X 0,Y 216.309,Z 507.926,A -85,B 0,C 180,E1 -20828.115,E2 -20828.115} C_VEL
LIN {X 0,Y 218.588,Z 502.001,A -85,B 0,C 180,E1 -20831.226,E2 -20831.226} C_VEL
LIN {X 0,Y 220.99,Z 495.583,A -85,B 0,C 180,E1 -20833.834,E2 -20833.834} C_VEL
LIN {X 0,Y 223.579,Z 488.024,A -85,B 0,C 180,E1 -20836.295,E2 -20836.295} C_VEL
LIN {X 0,Y 226.544,Z 478.659,A -85,B 0,C 180,E1 -20838.693,E2 -20838.693} C_VEL
LIN {X 0,Y 229.67,Z 467.69,A -85,B 0,C 180,E1 -20840.887,E2 -20840.887} C_VEL
LIN {X 0,Y 230.088,Z 464.666,A -85,B 0,C 180,E1 -20841.455,E2 -20841.455} C_VEL
LIN {X 0,Y 228.786,Z 455.28,A -85,B 0,C 180,E1 -20843.474,E2 -20843.474} C_VEL
LIN {X 0,Y 226.409,Z 445.271,A -85,B 0,C 180,E1 -20845.522,E2 -20845.522} C_VEL
LIN {X 0,Y 222.87,Z 435.027,A -85,B 0,C 180,E1 -20847.583,E2 -20847.583} C_VEL
LIN {X 0,Y 218.48,Z 425.428,A -85,B 0,C 180,E1 -20849.56,E2 -20849.56} C_VEL
LIN {X 0,Y 216.028,Z 421.015,A -85,B 0,C 180,E1 -20850.524,E2 -20850.524} C_VEL
LIN {X 0,Y 214.46,Z 418.105,A -85,B 0,C 180,E1 -20851.138,E2 -20851.138} C_VEL
LIN {X 0,Y 214.247,Z 417.206,A -85,B 0,C 180,E1 -20851.3,E2 -20851.3} C_VEL
LIN {X 0,Y 214.103,Z 415.801,A -85,B 0,C 180,E1 -20854.74,E2 -20854.74} C_VEL
LIN {X 0,Y 213.935,Z 414.276,A -85,B 0,C 180,E1 -20858.816,E2 -20858.816} C_VEL
LIN {X 0,Y 213.924,Z 413.835,A -85,B 0,C 180,E1 -20862.297,E2 -20862.297} C_VEL
LIN {X 0,Y 213.937,Z 413.832,A -85,B 0,C 180,E1 -20866.706,E2 -20866.706} C_VEL
LIN {X 0,Y 214.151,Z 413.805,A -85,B 0,C 180,E1 -20870.556,E2 -20870.556} C_VEL
LIN {X 0,Y 214.211,Z 413.797,A -85,B 0,C 180,E1 -20872.459,E2 -20872.459} C_VEL
LIN {X 0,Y 214.43,Z 413.776,A -85,B 0,C 180,E1 -20878.122,E2 -20878.122} C_VEL
LIN {X 0,Y 214.538,Z 413.762,A -85,B 0,C 180,E1 -20880,E2 -20880} C_VEL
LIN {X 0,Y 214.464,Z 413.771,A -85,B 0,C 180,E1 -20881.878,E2 -20881.878} C_VEL
LIN {X 0,Y 214.211,Z 413.801,A -85,B 0,C 180,E1 -20887.541,E2 -20887.541} C_VEL
LIN {X 0,Y 214.028,Z 413.825,A -85,B 0,C 180,E1 -20891.363,E2 -20891.363} C_VEL
LIN {X 0,Y 213.921,Z 413.839,A -85,B 0,C 180,E1 -20895.238,E2 -20895.238} C_VEL
LIN {X 0,Y 213.87,Z 413.846,A -85,B 0,C 180,E1 -20899.185,E2 -20899.185} C_VEL
LIN {X 0,Y 213.879,Z 414.113,A -85,B 0,C 180,E1 -20903.224,E2 -20903.224} C_VEL
LIN {X 0,Y 214.183,Z 416.106,A -85,B 0,C 180,E1 -20907.641,E2 -20907.641} C_VEL
LIN {X 0,Y 214.562,Z 418.22,A -85,B 0,C 180,E1 -20911.619,E2 -20911.619} C_VEL
LIN {X 0,Y 215.034,Z 420.938,A -85,B 0,C 180,E1 -20916.037,E2 -20916.037} C_VEL
LIN {X 0,Y 215.628,Z 424.232,A -85,B 0,C 180,E1 -20920.683,E2 -20920.683} C_VEL
LIN {X 0,Y 216.37,Z 428.157,A -85,B 0,C 180,E1 -20925.61,E2 -20925.61} C_VEL
LIN {X 0,Y 216.984,Z 431.707,A -85,B 0,C 180,E1 -20929.63,E2 -20929.63} C_VEL
LIN {X 0,Y 216.975,Z 434.354,A -85,B 0,C 180,E1 -20932.357,E2 -20932.357} C_VEL
LIN {X 0,Y 218.006,Z 437.737,A -85,B 0,C 180,E1 -20932.812,E2 -20932.812} C_VEL
LIN {X 0,Y 218.903,Z 440.003,A -85,B 0,C 180,E1 -20933.179,E2 -20933.179} C_VEL
LIN {X 0,Y 221.959,Z 450.444,A -85,B 0,C 180,E1 -20934.738,E2 -20934.738} C_VEL
LIN {X 0,Y 224.404,Z 462.24,A -85,B 0,C 180,E1 -20936.546,E2 -20936.546} C_VEL
LIN {X 0,Y 225.651,Z 473.817,A -85,B 0,C 180,E1 -20938.422,E2 -20938.422} C_VEL
LIN {X 0,Y 225.947,Z 484.993,A -85,B 0,C 180,E1 -20940.425,E2 -20940.425} C_VEL
LIN {X 0,Y 225.147,Z 495.728,A -85,B 0,C 180,E1 -20942.59,E2 -20942.59} C_VEL
LIN {X 0,Y 224.234,Z 501.841,A -85,B 0,C 180,E1 -20943.978,E2 -20943.978} C_VEL
LIN {X 0,Y 223.687,Z 503.561,A -85,B 0,C 180,E1 -20944.359,E2 -20944.359} C_VEL
LIN {X 0,Y 221.746,Z 507.781,A -85,B 0,C 180,E1 -20945.296,E2 -20945.296} C_VEL
LIN {X 0,Y 217.027,Z 514.214,A -85,B 0,C 180,E1 -20946.826,E2 -20946.826} C_VEL
LIN {X 0,Y 212.374,Z 520.077,A -85,B 0,C 180,E1 -20948.556,E2 -20948.556} C_VEL
LIN {X 0,Y 210.572,Z 523.325,A -85,B 0,C 180,E1 -20949.79,E2 -20949.79} C_VEL
LIN {X 0,Y 208.497,Z 528.822,A -85,B 0,C 180,E1 -20952.344,E2 -20952.344} C_VEL
LIN {X 0,Y 206.726,Z 533.748,A -85,B 0,C 180,E1 -20955.232,E2 -20955.232} C_VEL
LIN {X 0,Y 205.567,Z 537.58,A -85,B 0,C 180,E1 -20958.167,E2 -20958.167} C_VEL
LIN {X 0,Y 205.082,Z 539.584,A -85,B 0,C 180,E1 -20960.138,E2 -20960.138} C_VEL
LIN {X 0,Y 204.736,Z 541.171,A -85,B 0,C 180,E1 -20962.112,E2 -20962.112} C_VEL
LIN {X 0,Y 204.546,Z 542.784,A -85,B 0,C 180,E1 -20965.147,E2 -20965.147} C_VEL
LIN {X 0,Y 204.657,Z 543.425,A -85,B 0,C 180,E1 -20968.036,E2 -20968.036} C_VEL
LIN {X 0,Y 204.741,Z 543.388,A -85,B 0,C 180,E1 -20970.004,E2 -20970.004} C_VEL
LIN {X 0,Y 204.702,Z 542.898,A -85,B 0,C 180,E1 -20971.971,E2 -20971.971} C_VEL
LIN {X 0,Y 204.631,Z 541.265,A -85,B 0,C 180,E1 -20975.123,E2 -20975.123} C_VEL
LIN {X 0,Y 204.933,Z 537.878,A -85,B 0,C 180,E1 -20978.881,E2 -20978.881} C_VEL
LIN {X 0,Y 205.585,Z 534.031,A -85,B 0,C 180,E1 -20981.84,E2 -20981.84} C_VEL
LIN {X 0,Y 206.71,Z 529.044,A -85,B 0,C 180,E1 -20984.777,E2 -20984.777} C_VEL
LIN {X 0,Y 208.321,Z 522.769,A -85,B 0,C 180,E1 -20987.679,E2 -20987.679} C_VEL
LIN {X 0,Y 210.081,Z 516.389,A -85,B 0,C 180,E1 -20990.044,E2 -20990.044} C_VEL
LIN {X 0,Y 212.041,Z 508.64,A -85,B 0,C 180,E1 -20992.409,E2 -20992.409} C_VEL
LIN {X 0,Y 214.471,Z 499.282,A -85,B 0,C 180,E1 -20994.699,E2 -20994.699} C_VEL
LIN {X 0,Y 215.055,Z 496.034,A -85,B 0,C 180,E1 -20995.403,E2 -20995.403} C_VEL
LIN {X 0,Y 215.318,Z 485.907,A -85,B 0,C 180,E1 -20997.46,E2 -20997.46} C_VEL
LIN {X 0,Y 214.885,Z 474.693,A -85,B 0,C 180,E1 -20999.383,E2 -20999.383} C_VEL
LIN {X 0,Y 213.654,Z 462.041,A -85,B 0,C 180,E1 -21001.212,E2 -21001.212} C_VEL
LIN {X 0,Y 211.523,Z 448.969,A -85,B 0,C 180,E1 -21002.805,E2 -21002.805} C_VEL
LIN {X 0,Y 208.66,Z 435.995,A -85,B 0,C 180,E1 -21004.162,E2 -21004.162} C_VEL
LIN {X 0,Y 209.542,Z 432.792,A -85,B 0,C 180,E1 -21007.14,E2 -21007.14} C_VEL
LIN {X 0,Y 209.529,Z 430.296,A -85,B 0,C 180,E1 -21009.594,E2 -21009.594} C_VEL
LIN {X 0,Y 208.875,Z 426.394,A -85,B 0,C 180,E1 -21013.663,E2 -21013.663} C_VEL
LIN {X 0,Y 208.117,Z 422.516,A -85,B 0,C 180,E1 -21017.986,E2 -21017.986} C_VEL
LIN {X 0,Y 207.446,Z 418.807,A -85,B 0,C 180,E1 -21022.423,E2 -21022.423} C_VEL
LIN {X 0,Y 206.822,Z 415.229,A -85,B 0,C 180,E1 -21027.064,E2 -21027.064} C_VEL
LIN {X 0,Y 206.75,Z 414.736,A -85,B 0,C 180,E1 -21028.051,E2 -21028.051} C_VEL
LIN {X 0,Y 206.774,Z 414.731,A -85,B 0,C 180,E1 -21032.099,E2 -21032.099} C_VEL
LIN {X 0,Y 206.795,Z 414.728,A -85,B 0,C 180,E1 -21036.585,E2 -21036.585} C_VEL
LIN {X 0,Y 206.883,Z 414.72,A -85,B 0,C 180,E1 -21042.197,E2 -21042.197} C_VEL
LIN {X 0,Y 206.904,Z 414.718,A -85,B 0,C 180,E1 -21046.245,E2 -21046.245} C_VEL
LIN {X 0,Y 207.11,Z 414.691,A -85,B 0,C 180,E1 -21050.231,E2 -21050.231} C_VEL
LIN {X 0,Y 207.069,Z 414.694,A -85,B 0,C 180,E1 -21054.156,E2 -21054.156} C_VEL
LIN {X 0,Y 207.389,Z 414.654,A -85,B 0,C 180,E1 -21058.058,E2 -21058.058} C_VEL
LIN {X 0,Y 207.52,Z 414.636,A -85,B 0,C 180,E1 -21060,E2 -21060} C_VEL
LIN {X 0,Y 207.39,Z 414.65,A -85,B 0,C 180,E1 -21061.942,E2 -21061.942} C_VEL
LIN {X 0,Y 207.177,Z 414.65,A -85,B 0,C 180,E1 -21067.798,E2 -21067.798} C_VEL
LIN {X 0,Y 206.991,Z 414.698,A -85,B 0,C 180,E1 -21071.754,E2 -21071.754} C_VEL
LIN {X 0,Y 206.875,Z 414.711,A -85,B 0,C 180,E1 -21075.77,E2 -21075.77} C_VEL
LIN {X 0,Y 206.793,Z 414.698,A -85,B 0,C 180,E1 -21079.868,E2 -21079.868} C_VEL
LIN {X 0,Y 206.773,Z 414.724,A -85,B 0,C 180,E1 -21084.071,E2 -21084.071} C_VEL
LIN {X 0,Y 206.746,Z 414.728,A -85,B 0,C 180,E1 -21088.418,E2 -21088.418} C_VEL
LIN {X 0,Y 206.707,Z 414.711,A -85,B 0,C 180,E1 -21092.956,E2 -21092.956} C_VEL
LIN {X 0,Y 206.688,Z 414.739,A -85,B 0,C 180,E1 -21097.738,E2 -21097.738} C_VEL
LIN {X 0,Y 206.65,Z 414.733,A -85,B 0,C 180,E1 -21101.561,E2 -21101.561} C_VEL
LIN {X 0,Y 206.642,Z 414.735,A -85,B 0,C 180,E1 -21105.579,E2 -21105.579} C_VEL
LIN {X 0,Y 206.668,Z 414.739,A -85,B 0,C 180,E1 -21109.747,E2 -21109.747} C_VEL
LIN {X 0,Y 206.706,Z 414.734,A -85,B 0,C 180,E1 -21114.686,E2 -21114.686} C_VEL
LIN {X 0,Y 206.729,Z 414.726,A -85,B 0,C 180,E1 -21119.336,E2 -21119.336} C_VEL
LIN {X 0,Y 206.739,Z 414.737,A -85,B 0,C 180,E1 -21123.769,E2 -21123.769} C_VEL
LIN {X 0,Y 206.764,Z 414.732,A -85,B 0,C 180,E1 -21128.04,E2 -21128.04} C_VEL
LIN {X 0,Y 206.878,Z 414.714,A -85,B 0,C 180,E1 -21132.193,E2 -21132.193} C_VEL
LIN {X 0,Y 206.819,Z 414.724,A -85,B 0,C 180,E1 -21136.236,E2 -21136.236} C_VEL
LIN {X 0,Y 206.751,Z 414.961,A -85,B 0,C 180,E1 -21138.725,E2 -21138.725} C_VEL
LIN {X 0,Y 206.747,Z 415.029,A -85,B 0,C 180,E1 -21138.824,E2 -21138.824} C_VEL
LIN {X 0,Y 207.915,Z 418.177,A -85,B 0,C 180,E1 -21139.214,E2 -21139.214} C_VEL
LIN {X 0,Y 211.767,Z 427.387,A -85,B 0,C 180,E1 -21140.524,E2 -21140.524} C_VEL
LIN {X 0,Y 214.513,Z 436.916,A -85,B 0,C 180,E1 -21141.888,E2 -21141.888} C_VEL
LIN {X 0,Y 217.284,Z 449.295,A -85,B 0,C 180,E1 -21143.911,E2 -21143.911} C_VEL
LIN {X 0,Y 219.163,Z 459.595,A -85,B 0,C 180,E1 -21145.859,E2 -21145.859} C_VEL
LIN {X 0,Y 219.3,Z 460.799,A -85,B 0,C 180,E1 -21146.091,E2 -21146.091} C_VEL
LIN {X 0,Y 216.866,Z 471.969,A -85,B 0,C 180,E1 -21148.139,E2 -21148.139} C_VEL
LIN {X 0,Y 214.367,Z 481.999,A -85,B 0,C 180,E1 -21150.466,E2 -21150.466} C_VEL
LIN {X 0,Y 212.194,Z 490.198,A -85,B 0,C 180,E1 -21152.844,E2 -21152.844} C_VEL
LIN {X 0,Y 209.931,Z 498.185,A -85,B 0,C 180,E1 -21155.76,E2 -21155.76} C_VEL
LIN {X 0,Y 208.097,Z 504.573,A -85,B 0,C 180,E1 -21158.738,E2 -21158.738} C_VEL
LIN {X 0,Y 206.724,Z 509.615,A -85,B 0,C 180,E1 -21161.766,E2 -21161.766} C_VEL
LIN {X 0,Y 205.67,Z 513.481,A -85,B 0,C 180,E1 -21164.845,E2 -21164.845} C_VEL
LIN {X 0,Y 204.912,Z 516.256,A -85,B 0,C 180,E1 -21167.975,E2 -21167.975} C_VEL
LIN {X 0,Y 204.628,Z 517.521,A -85,B 0,C 180,E1 -21170.083,E2 -21170.083} C_VEL
LIN {X 0,Y 204.504,Z 518.31,A -85,B 0,C 180,E1 -21172.207,E2 -21172.207} C_VEL
LIN {X 0,Y 204.593,Z 518.67,A -85,B 0,C 180,E1 -21174.339,E2 -21174.339} C_VEL
LIN {X 0,Y 204.862,Z 518.468,A -85,B 0,C 180,E1 -21176.88,E2 -21176.88} C_VEL
LIN {X 0,Y 205.801,Z 516.899,A -85,B 0,C 180,E1 -21180.808,E2 -21180.808} C_VEL
LIN {X 0,Y 206.994,Z 514.326,A -85,B 0,C 180,E1 -21184.066,E2 -21184.066} C_VEL
LIN {X 0,Y 208.661,Z 510.49,A -85,B 0,C 180,E1 -21187.314,E2 -21187.314} C_VEL
LIN {X 0,Y 210.901,Z 505.155,A -85,B 0,C 180,E1 -21190.59,E2 -21190.59} C_VEL
LIN {X 0,Y 213.622,Z 498.456,A -85,B 0,C 180,E1 -21193.694,E2 -21193.694} C_VEL
LIN {X 0,Y 216.727,Z 490.003,A -85,B 0,C 180,E1 -21196.676,E2 -21196.676} C_VEL
LIN {X 0,Y 219.361,Z 482.276,A -85,B 0,C 180,E1 -21198.836,E2 -21198.836} C_VEL
LIN {X 0,Y 222.32,Z 472.89,A -85,B 0,C 180,E1 -21200.94,E2 -21200.94} C_VEL
LIN {X 0,Y 223.59,Z 468.421,A -85,B 0,C 180,E1 -21201.789,E2 -21201.789} C_VEL
LIN {X 0,Y 223.707,Z 465.199,A -85,B 0,C 180,E1 -21202.482,E2 -21202.482} C_VEL
LIN {X 0,Y 222.268,Z 455.173,A -85,B 0,C 180,E1 -21204.756,E2 -21204.756} C_VEL
LIN {X 0,Y 219.927,Z 445.825,A -85,B 0,C 180,E1 -21206.794,E2 -21206.794} C_VEL
LIN {X 0,Y 216.782,Z 436.791,A -85,B 0,C 180,E1 -21208.754,E2 -21208.754} C_VEL
LIN {X 0,Y 213.127,Z 428.919,A -85,B 0,C 180,E1 -21210.558,E2 -21210.558} C_VEL
LIN {X 0,Y 211.477,Z 425.749,A -85,B 0,C 180,E1 -21211.286,E2 -21211.286} C_VEL
LIN {X 0,Y 209.406,Z 422.073,A -85,B 0,C 180,E1 -21212.176,E2 -21212.176} C_VEL
LIN {X 0,Y 207.569,Z 419.076,A -85,B 0,C 180,E1 -21212.937,E2 -21212.937} C_VEL
LIN {X 0,Y 207.235,Z 417.815,A -85,B 0,C 180,E1 -21213.162,E2 -21213.162} C_VEL
LIN {X 0,Y 207.004,Z 416.023,A -85,B 0,C 180,E1 -21218.071,E2 -21218.071} C_VEL
LIN {X 0,Y 206.87,Z 414.714,A -85,B 0,C 180,E1 -21222.196,E2 -21222.196} C_VEL
LIN {X 0,Y 206.88,Z 414.713,A -85,B 0,C 180,E1 -21226.243,E2 -21226.243} C_VEL
LIN {X 0,Y 207.089,Z 414.684,A -85,B 0,C 180,E1 -21230.231,E2 -21230.231} C_VEL
LIN {X 0,Y 207.058,Z 414.691,A -85,B 0,C 180,E1 -21234.156,E2 -21234.156} C_VEL
LIN {X 0,Y 207.367,Z 414.656,A -85,B 0,C 180,E1 -21238.058,E2 -21238.058} C_VEL
LIN {X 0,Y 207.502,Z 414.638,A -85,B 0,C 180,E1 -21240,E2 -21240} C_VEL
LIN {X 0,Y 207.397,Z 414.651,A -85,B 0,C 180,E1 -21241.942,E2 -21241.942} C_VEL
LIN {X 0,Y 207.151,Z 414.681,A -85,B 0,C 180,E1 -21247.8,E2 -21247.8} C_VEL
LIN {X 0,Y 206.965,Z 414.706,A -85,B 0,C 180,E1 -21251.756,E2 -21251.756} C_VEL
LIN {X 0,Y 206.861,Z 414.717,A -85,B 0,C 180,E1 -21255.771,E2 -21255.771} C_VEL
LIN {X 0,Y 206.809,Z 414.727,A -85,B 0,C 180,E1 -21259.867,E2 -21259.867} C_VEL
LIN {X 0,Y 207.035,Z 416.187,A -85,B 0,C 180,E1 -21264.039,E2 -21264.039} C_VEL
LIN {X 0,Y 207.329,Z 418.126,A -85,B 0,C 180,E1 -21268.332,E2 -21268.332} C_VEL
LIN {X 0,Y 207.732,Z 420.499,A -85,B 0,C 180,E1 -21272.773,E2 -21272.773} C_VEL
LIN {X 0,Y 208.253,Z 423.399,A -85,B 0,C 180,E1 -21277.406,E2 -21277.406} C_VEL
LIN {X 0,Y 208.859,Z 426.876,A -85,B 0,C 180,E1 -21282.299,E2 -21282.299} C_VEL
LIN {X 0,Y 209.319,Z 429.114,A -85,B 0,C 180,E1 -21285.17,E2 -21285.17} C_VEL
LIN {X 0,Y 209.916,Z 432.567,A -85,B 0,C 180,E1 -21289.235,E2 -21289.235} C_VEL
LIN {X 0,Y 210.09,Z 433.972,A -85,B 0,C 180,E1 -21290.607,E2 -21290.607} C_VEL
LIN {X 0,Y 211.272,Z 437.404,A -85,B 0,C 180,E1 -21291.15,E2 -21291.15} C_VEL
LIN {X 0,Y 212.372,Z 439.614,A -85,B 0,C 180,E1 -21291.592,E2 -21291.592} C_VEL
LIN {X 0,Y 214.948,Z 447.294,A -85,B 0,C 180,E1 -21292.875,E2 -21292.875} C_VEL
LIN {X 0,Y 217.779,Z 459.875,A -85,B 0,C 180,E1 -21294.932,E2 -21294.932} C_VEL
LIN {X 0,Y 219.187,Z 470.514,A -85,B 0,C 180,E1 -21296.732,E2 -21296.732} C_VEL
LIN {X 0,Y 219.652,Z 481.714,A -85,B 0,C 180,E1 -21298.776,E2 -21298.776} C_VEL
LIN {X 0,Y 219.243,Z 491.287,A -85,B 0,C 180,E1 -21300.711,E2 -21300.711} C_VEL
LIN {X 0,Y 218.216,Z 499.983,A -85,B 0,C 180,E1 -21302.686,E2 -21302.686} C_VEL
LIN {X 0,Y 216.628,Z 505.574,A -85,B 0,C 180,E1 -21304.03,E2 -21304.03} C_VEL
LIN {X 0,Y 213.805,Z 513.598,A -85,B 0,C 180,E1 -21306.259,E2 -21306.259} C_VEL
LIN {X 0,Y 211.267,Z 521.109,A -85,B 0,C 180,E1 -21308.876,E2 -21308.876} C_VEL
LIN {X 0,Y 210.572,Z 523.325,A -85,B 0,C 180,E1 -21309.79,E2 -21309.79} C_VEL
LIN {X 0,Y 208.793,Z 526.392,A -85,B 0,C 180,E1 -21311.085,E2 -21311.085} C_VEL
LIN {X 0,Y 204.316,Z 530.863,A -85,B 0,C 180,E1 -21313.207,E2 -21313.207} C_VEL
LIN {X 0,Y 200.115,Z 534.617,A -85,B 0,C 180,E1 -21315.519,E2 -21315.519} C_VEL
LIN {X 0,Y 198.807,Z 536.547,A -85,B 0,C 180,E1 -21317.076,E2 -21317.076} C_VEL
LIN {X 0,Y 198.045,Z 539.267,A -85,B 0,C 180,E1 -21319.784,E2 -21319.784} C_VEL
LIN {X 0,Y 197.684,Z 540.815,A -85,B 0,C 180,E1 -21321.829,E2 -21321.829} C_VEL
LIN {X 0,Y 197.462,Z 542.658,A -85,B 0,C 180,E1 -21325.922,E2 -21325.922} C_VEL
LIN {X 0,Y 197.566,Z 543.001,A -85,B 0,C 180,E1 -21327.965,E2 -21327.965} C_VEL
LIN {X 0,Y 197.673,Z 542.936,A -85,B 0,C 180,E1 -21330.004,E2 -21330.004} C_VEL
LIN {X 0,Y 197.611,Z 542.415,A -85,B 0,C 180,E1 -21332.042,E2 -21332.042} C_VEL
LIN {X 0,Y 197.541,Z 540.95,A -85,B 0,C 180,E1 -21335.014,E2 -21335.014} C_VEL
LIN {X 0,Y 197.907,Z 537.313,A -85,B 0,C 180,E1 -21339.199,E2 -21339.199} C_VEL
LIN {X 0,Y 198.598,Z 533.417,A -85,B 0,C 180,E1 -21342.263,E2 -21342.263} C_VEL
LIN {X 0,Y 199.82,Z 528.382,A -85,B 0,C 180,E1 -21345.299,E2 -21345.299} C_VEL
LIN {X 0,Y 201.522,Z 522.045,A -85,B 0,C 180,E1 -21348.296,E2 -21348.296} C_VEL
LIN {X 0,Y 203.019,Z 516.937,A -85,B 0,C 180,E1 -21350.257,E2 -21350.257} C_VEL
LIN {X 0,Y 204.985,Z 509.418,A -85,B 0,C 180,E1 -21352.692,E2 -21352.692} C_VEL
LIN {X 0,Y 207.495,Z 500.348,A -85,B 0,C 180,E1 -21355.052,E2 -21355.052} C_VEL
LIN {X 0,Y 208.259,Z 496.093,A -85,B 0,C 180,E1 -21356.025,E2 -21356.025} C_VEL
LIN {X 0,Y 208.576,Z 484.991,A -85,B 0,C 180,E1 -21358.356,E2 -21358.356} C_VEL
LIN {X 0,Y 208.111,Z 473.154,A -85,B 0,C 180,E1 -21360.438,E2 -21360.438} C_VEL
LIN {X 0,Y 206.835,Z 460.651,A -85,B 0,C 180,E1 -21362.304,E2 -21362.304} C_VEL
LIN {X 0,Y 204.668,Z 447.805,A -85,B 0,C 180,E1 -21363.92,E2 -21363.92} C_VEL
LIN {X 0,Y 201.906,Z 435.614,A -85,B 0,C 180,E1 -21365.243,E2 -21365.243} C_VEL
LIN {X 0,Y 202.419,Z 433.772,A -85,B 0,C 180,E1 -21367.006,E2 -21367.006} C_VEL
LIN {X 0,Y 202.552,Z 432.121,A -85,B 0,C 180,E1 -21368.653,E2 -21368.653} C_VEL
LIN {X 0,Y 201.941,Z 428.019,A -85,B 0,C 180,E1 -21373.042,E2 -21373.042} C_VEL
LIN {X 0,Y 201.262,Z 424.394,A -85,B 0,C 180,E1 -21377.169,E2 -21377.169} C_VEL
LIN {X 0,Y 200.649,Z 421.294,A -85,B 0,C 180,E1 -21380.915,E2 -21380.915} C_VEL
LIN {X 0,Y 200.006,Z 417.542,A -85,B 0,C 180,E1 -21385.79,E2 -21385.79} C_VEL
LIN {X 0,Y 199.676,Z 415.617,A -85,B 0,C 180,E1 -21388.724,E2 -21388.724} C_VEL
LIN {X 0,Y 199.695,Z 415.61,A -85,B 0,C 180,E1 -21392.773,E2 -21392.773} C_VEL
LIN {X 0,Y 199.748,Z 415.604,A -85,B 0,C 180,E1 -21397.23,E2 -21397.23} C_VEL
LIN {X 0,Y 199.807,Z 415.601,A -85,B 0,C 180,E1 -21401.758,E2 -21401.758} C_VEL
LIN {X 0,Y 199.845,Z 415.596,A -85,B 0,C 180,E1 -21405.749,E2 -21405.749} C_VEL
LIN {X 0,Y 200.033,Z 415.572,A -85,B 0,C 180,E1 -21409.882,E2 -21409.882} C_VEL
LIN {X 0,Y 200.031,Z 415.571,A -85,B 0,C 180,E1 -21413.949,E2 -21413.949} C_VEL
LIN {X 0,Y 200.329,Z 415.533,A -85,B 0,C 180,E1 -21417.989,E2 -21417.989} C_VEL
LIN {X 0,Y 200.485,Z 415.513,A -85,B 0,C 180,E1 -21420,E2 -21420} C_VEL
LIN {X 0,Y 200.037,Z 415.554,A -85,B 0,C 180,E1 -21424.029,E2 -21424.029} C_VEL
LIN {X 0,Y 200.121,Z 415.53,A -85,B 0,C 180,E1 -21428.075,E2 -21428.075} C_VEL
LIN {X 0,Y 199.923,Z 415.582,A -85,B 0,C 180,E1 -21432.176,E2 -21432.176} C_VEL
LIN {X 0,Y 199.813,Z 415.587,A -85,B 0,C 180,E1 -21436.343,E2 -21436.343} C_VEL
LIN {X 0,Y 199.709,Z 415.579,A -85,B 0,C 180,E1 -21440.604,E2 -21440.604} C_VEL
LIN {X 0,Y 199.682,Z 415.608,A -85,B 0,C 180,E1 -21444.983,E2 -21444.983} C_VEL
LIN {X 0,Y 199.674,Z 415.604,A -85,B 0,C 180,E1 -21449.522,E2 -21449.522} C_VEL
LIN {X 0,Y 199.68,Z 415.585,A -85,B 0,C 180,E1 -21452.354,E2 -21452.354} C_VEL
LIN {X 0,Y 199.632,Z 415.614,A -85,B 0,C 180,E1 -21456.761,E2 -21456.761} C_VEL
LIN {X 0,Y 199.617,Z 415.62,A -85,B 0,C 180,E1 -21459.326,E2 -21459.326} C_VEL
LIN {X 0,Y 199.583,Z 415.61,A -85,B 0,C 180,E1 -21462.308,E2 -21462.308} C_VEL
LIN {X 0,Y 199.588,Z 415.609,A -85,B 0,C 180,E1 -21465.227,E2 -21465.227} C_VEL
LIN {X 0,Y 199.588,Z 415.623,A -85,B 0,C 180,E1 -21468.003,E2 -21468.003} C_VEL
LIN {X 0,Y 199.618,Z 415.613,A -85,B 0,C 180,E1 -21470.765,E2 -21470.765} C_VEL
LIN {X 0,Y 199.621,Z 415.621,A -85,B 0,C 180,E1 -21475.711,E2 -21475.711} C_VEL
LIN {X 0,Y 199.707,Z 415.609,A -85,B 0,C 180,E1 -21478.134,E2 -21478.134} C_VEL
LIN {X 0,Y 199.694,Z 415.616,A -85,B 0,C 180,E1 -21482.769,E2 -21482.769} C_VEL
LIN {X 0,Y 199.744,Z 415.604,A -85,B 0,C 180,E1 -21487.226,E2 -21487.226} C_VEL
LIN {X 0,Y 199.801,Z 415.594,A -85,B 0,C 180,E1 -21491.754,E2 -21491.754} C_VEL
LIN {X 0,Y 199.732,Z 415.607,A -85,B 0,C 180,E1 -21496.775,E2 -21496.775} C_VEL
LIN {X 0,Y 199.714,Z 415.609,A -85,B 0,C 180,E1 -21497.614,E2 -21497.614} C_VEL
LIN {X 0,Y 200.791,Z 418.593,A -85,B 0,C 180,E1 -21498.037,E2 -21498.037} C_VEL
LIN {X 0,Y 205.103,Z 428.488,A -85,B 0,C 180,E1 -21499.57,E2 -21499.57} C_VEL
LIN {X 0,Y 207.923,Z 437.66,A -85,B 0,C 180,E1 -21500.99,E2 -21500.99} C_VEL
LIN {X 0,Y 210.49,Z 449.369,A -85,B 0,C 180,E1 -21502.968,E2 -21502.968} C_VEL
LIN {X 0,Y 212.497,Z 460.911,A -85,B 0,C 180,E1 -21505.233,E2 -21505.233} C_VEL
LIN {X 0,Y 212.638,Z 462.163,A -85,B 0,C 180,E1 -21505.494,E2 -21505.494} C_VEL
LIN {X 0,Y 210.093,Z 473.218,A -85,B 0,C 180,E1 -21507.616,E2 -21507.616} C_VEL
LIN {X 0,Y 207.536,Z 483.053,A -85,B 0,C 180,E1 -21509.996,E2 -21509.996} C_VEL
LIN {X 0,Y 204.925,Z 492.262,A -85,B 0,C 180,E1 -21512.842,E2 -21512.842} C_VEL
LIN {X 0,Y 202.587,Z 500.184,A -85,B 0,C 180,E1 -21515.97,E2 -21515.97} C_VEL
LIN {X 0,Y 200.808,Z 506.267,A -85,B 0,C 180,E1 -21519.057,E2 -21519.057} C_VEL
LIN {X 0,Y 199.438,Z 511.023,A -85,B 0,C 180,E1 -21522.202,E2 -21522.202} C_VEL
LIN {X 0,Y 198.426,Z 514.628,A -85,B 0,C 180,E1 -21525.401,E2 -21525.401} C_VEL
LIN {X 0,Y 197.701,Z 517.164,A -85,B 0,C 180,E1 -21528.655,E2 -21528.655} C_VEL
LIN {X 0,Y 197.422,Z 518.732,A -85,B 0,C 180,E1 -21532.246,E2 -21532.246} C_VEL
LIN {X 0,Y 197.559,Z 519.113,A -85,B 0,C 180,E1 -21535.265,E2 -21535.265} C_VEL
LIN {X 0,Y 197.873,Z 518.837,A -85,B 0,C 180,E1 -21537.494,E2 -21537.494} C_VEL
LIN {X 0,Y 198.387,Z 518.11,A -85,B 0,C 180,E1 -21539.728,E2 -21539.728} C_VEL
LIN {X 0,Y 199.117,Z 516.756,A -85,B 0,C 180,E1 -21542.103,E2 -21542.103} C_VEL
LIN {X 0,Y 200.461,Z 514.011,A -85,B 0,C 180,E1 -21545.338,E2 -21545.338} C_VEL
LIN {X 0,Y 202.386,Z 509.91,A -85,B 0,C 180,E1 -21548.681,E2 -21548.681} C_VEL
LIN {X 0,Y 204.828,Z 504.368,A -85,B 0,C 180,E1 -21551.99,E2 -21551.99} C_VEL
LIN {X 0,Y 207.902,Z 497.108,A -85,B 0,C 180,E1 -21555.22,E2 -21555.22} C_VEL
LIN {X 0,Y 210.752,Z 489.65,A -85,B 0,C 180,E1 -21557.824,E2 -21557.824} C_VEL
LIN {X 0,Y 213.818,Z 481.112,A -85,B 0,C 180,E1 -21560.196,E2 -21560.196} C_VEL
LIN {X 0,Y 216.945,Z 471.377,A -85,B 0,C 180,E1 -21562.326,E2 -21562.326} C_VEL
LIN {X 0,Y 217.578,Z 468.324,A -85,B 0,C 180,E1 -21562.959,E2 -21562.959} C_VEL
LIN {X 0,Y 216.396,Z 458.358,A -85,B 0,C 180,E1 -21565.377,E2 -21565.377} C_VEL
LIN {X 0,Y 214.03,Z 448.217,A -85,B 0,C 180,E1 -21567.752,E2 -21567.752} C_VEL
LIN {X 0,Y 211.325,Z 440.066,A -85,B 0,C 180,E1 -21569.663,E2 -21569.663} C_VEL
LIN {X 0,Y 206.975,Z 430.562,A -85,B 0,C 180,E1 -21572.025,E2 -21572.025} C_VEL
LIN {X 0,Y 204.894,Z 426.809,A -85,B 0,C 180,E1 -21573.025,E2 -21573.025} C_VEL
LIN {X 0,Y 202.728,Z 423.031,A -85,B 0,C 180,E1 -21574.045,E2 -21574.045} C_VEL
LIN {X 0,Y 200.77,Z 420.395,A -85,B 0,C 180,E1 -21574.885,E2 -21574.885} C_VEL
LIN {X 0,Y 200.123,Z 418.453,A -85,B 0,C 180,E1 -21575.29,E2 -21575.29} C_VEL
LIN {X 0,Y 199.968,Z 417.069,A -85,B 0,C 180,E1 -21579.424,E2 -21579.424} C_VEL
LIN {X 0,Y 199.831,Z 415.866,A -85,B 0,C 180,E1 -21583.659,E2 -21583.659} C_VEL
LIN {X 0,Y 199.87,Z 415.586,A -85,B 0,C 180,E1 -21587.821,E2 -21587.821} C_VEL
LIN {X 0,Y 200.095,Z 415.558,A -85,B 0,C 180,E1 -21591.924,E2 -21591.924} C_VEL
LIN {X 0,Y 200.307,Z 415.536,A -85,B 0,C 180,E1 -21597.989,E2 -21597.989} C_VEL
LIN {X 0,Y 200.466,Z 415.515,A -85,B 0,C 180,E1 -21600,E2 -21600} C_VEL
LIN {X 0,Y 200.334,Z 415.53,A -85,B 0,C 180,E1 -21602.011,E2 -21602.011} C_VEL
LIN {X 0,Y 200.095,Z 415.561,A -85,B 0,C 180,E1 -21608.077,E2 -21608.077} C_VEL
LIN {X 0,Y 199.898,Z 415.585,A -85,B 0,C 180,E1 -21612.178,E2 -21612.178} C_VEL
LIN {X 0,Y 199.799,Z 415.598,A -85,B 0,C 180,E1 -21616.344,E2 -21616.344} C_VEL
LIN {X 0,Y 199.852,Z 415.934,A -85,B 0,C 180,E1 -21618.451,E2 -21618.451} C_VEL
LIN {X 0,Y 200.166,Z 417.914,A -85,B 0,C 180,E1 -21624.105,E2 -21624.105} C_VEL
LIN {X 0,Y 200.488,Z 420.313,A -85,B 0,C 180,E1 -21629.391,E2 -21629.391} C_VEL
LIN {X 0,Y 200.915,Z 422.844,A -85,B 0,C 180,E1 -21634.034,E2 -21634.034} C_VEL
LIN {X 0,Y 201.227,Z 424.352,A -85,B 0,C 180,E1 -21636.563,E2 -21636.563} C_VEL
LIN {X 0,Y 201.596,Z 426.587,A -85,B 0,C 180,E1 -21639.926,E2 -21639.926} C_VEL
LIN {X 0,Y 202.146,Z 429.607,A -85,B 0,C 180,E1 -21644.055,E2 -21644.055} C_VEL
LIN {X 0,Y 202.831,Z 433.321,A -85,B 0,C 180,E1 -21648.515,E2 -21648.515} C_VEL
LIN {X 0,Y 204.042,Z 436.535,A -85,B 0,C 180,E1 -21649.105,E2 -21649.105} C_VEL
LIN {X 0,Y 205.672,Z 439.072,A -85,B 0,C 180,E1 -21649.775,E2 -21649.775} C_VEL
LIN {X 0,Y 208.749,Z 447.333,A -85,B 0,C 180,E1 -21651.376,E2 -21651.376} C_VEL
LIN {X 0,Y 211.242,Z 457.844,A -85,B 0,C 180,E1 -21653.217,E2 -21653.217} C_VEL
LIN {X 0,Y 212.726,Z 467.711,A -85,B 0,C 180,E1 -21654.991,E2 -21654.991} C_VEL
LIN {X 0,Y 213.411,Z 479.036,A -85,B 0,C 180,E1 -21657.124,E2 -21657.124} C_VEL
LIN {X 0,Y 213.167,Z 489.179,A -85,B 0,C 180,E1 -21659.222,E2 -21659.222} C_VEL
LIN {X 0,Y 212.083,Z 498.189,A -85,B 0,C 180,E1 -21661.287,E2 -21661.287} C_VEL
LIN {X 0,Y 210.917,Z 503.874,A -85,B 0,C 180,E1 -21662.736,E2 -21662.736} C_VEL
LIN {X 0,Y 207.32,Z 513.576,A -85,B 0,C 180,E1 -21665.469,E2 -21665.469} C_VEL
LIN {X 0,Y 204.451,Z 521.482,A -85,B 0,C 180,E1 -21668.361,E2 -21668.361} C_VEL
LIN {X 0,Y 202.402,Z 526.76,A -85,B 0,C 180,E1 -21670.744,E2 -21670.744} C_VEL
LIN {X 0,Y 200.411,Z 532.031,A -85,B 0,C 180,E1 -21673.712,E2 -21673.712} C_VEL
LIN {X 0,Y 198.807,Z 536.547,A -85,B 0,C 180,E1 -21677.076,E2 -21677.076} C_VEL
LIN {X 0,Y 197.652,Z 538.262,A -85,B 0,C 180,E1 -21678.68,E2 -21678.68} C_VEL
LIN {X 0,Y 194.25,Z 540.42,A -85,B 0,C 180,E1 -21681.327,E2 -21681.327} C_VEL
LIN {X 0,Y 191.594,Z 541.615,A -85,B 0,C 180,E1 -21683.532,E2 -21683.532} C_VEL
LIN {X 0,Y 190.476,Z 542.161,A -85,B 0,C 180,E1 -21685.274,E2 -21685.274} C_VEL
LIN {X 0,Y 190.383,Z 542.271,A -85,B 0,C 180,E1 -21685.868,E2 -21685.868} C_VEL
LIN {X 0,Y 190.478,Z 542.578,A -85,B 0,C 180,E1 -21687.89,E2 -21687.89} C_VEL
LIN {X 0,Y 190.606,Z 542.473,A -85,B 0,C 180,E1 -21690.004,E2 -21690.004} C_VEL
LIN {X 0,Y 190.523,Z 541.927,A -85,B 0,C 180,E1 -21692.118,E2 -21692.118} C_VEL
LIN {X 0,Y 190.461,Z 540.602,A -85,B 0,C 180,E1 -21694.926,E2 -21694.926} C_VEL
LIN {X 0,Y 190.704,Z 537.806,A -85,B 0,C 180,E1 -21698.481,E2 -21698.481} C_VEL
LIN {X 0,Y 191.31,Z 534.225,A -85,B 0,C 180,E1 -21701.661,E2 -21701.661} C_VEL
LIN {X 0,Y 192.396,Z 529.518,A -85,B 0,C 180,E1 -21704.819,E2 -21704.819} C_VEL
LIN {X 0,Y 194.134,Z 523.563,A -85,B 0,C 180,E1 -21707.925,E2 -21707.925} C_VEL
LIN {X 0,Y 196.269,Z 516.12,A -85,B 0,C 180,E1 -21710.986,E2 -21710.986} C_VEL
LIN {X 0,Y 198.866,Z 506.856,A -85,B 0,C 180,E1 -21713.983,E2 -21713.983} C_VEL
LIN {X 0,Y 201.406,Z 497.231,A -85,B 0,C 180,E1 -21716.421,E2 -21716.421} C_VEL
LIN {X 0,Y 201.854,Z 487.531,A -85,B 0,C 180,E1 -21718.607,E2 -21718.607} C_VEL
LIN {X 0,Y 201.644,Z 476.993,A -85,B 0,C 180,E1 -21720.649,E2 -21720.649} C_VEL
LIN {X 0,Y 200.79,Z 465.848,A -85,B 0,C 180,E1 -21722.498,E2 -21722.498} C_VEL
LIN {X 0,Y 199.099,Z 453.453,A -85,B 0,C 180,E1 -21724.254,E2 -21724.254} C_VEL
LIN {X 0,Y 196.324,Z 440.372,A -85,B 0,C 180,E1 -21725.844,E2 -21725.844} C_VEL
LIN {X 0,Y 195.147,Z 435.19,A -85,B 0,C 180,E1 -21726.398,E2 -21726.398} C_VEL
LIN {X 0,Y 195.463,Z 432.694,A -85,B 0,C 180,E1 -21728.997,E2 -21728.997} C_VEL
LIN {X 0,Y 194.887,Z 428.849,A -85,B 0,C 180,E1 -21733.254,E2 -21733.254} C_VEL
LIN {X 0,Y 194.119,Z 424.876,A -85,B 0,C 180,E1 -21737.949,E2 -21737.949} C_VEL
LIN {X 0,Y 193.356,Z 420.827,A -85,B 0,C 180,E1 -21743.101,E2 -21743.101} C_VEL
LIN {X 0,Y 192.897,Z 418.088,A -85,B 0,C 180,E1 -21746.933,E2 -21746.933} C_VEL
LIN {X 0,Y 192.627,Z 416.495,A -85,B 0,C 180,E1 -21749.539,E2 -21749.539} C_VEL
LIN {X 0,Y 192.67,Z 416.488,A -85,B 0,C 180,E1 -21751.693,E2 -21751.693} C_VEL
LIN {X 0,Y 192.716,Z 416.481,A -85,B 0,C 180,E1 -21756.35,E2 -21756.35} C_VEL
LIN {X 0,Y 192.742,Z 416.481,A -85,B 0,C 180,E1 -21761.458,E2 -21761.458} C_VEL
LIN {X 0,Y 192.773,Z 416.477,A -85,B 0,C 180,E1 -21765.214,E2 -21765.214} C_VEL
LIN {X 0,Y 192.956,Z 416.453,A -85,B 0,C 180,E1 -21769.567,E2 -21769.567} C_VEL
LIN {X 0,Y 192.993,Z 416.447,A -85,B 0,C 180,E1 -21773.728,E2 -21773.728} C_VEL
LIN {X 0,Y 193.271,Z 416.412,A -85,B 0,C 180,E1 -21777.916,E2 -21777.916} C_VEL
LIN {X 0,Y 193.45,Z 416.389,A -85,B 0,C 180,E1 -21780,E2 -21780} C_VEL
LIN {X 0,Y 192.983,Z 416.431,A -85,B 0,C 180,E1 -21784.177,E2 -21784.177} C_VEL
LIN {X 0,Y 193.072,Z 416.409,A -85,B 0,C 180,E1 -21788.372,E2 -21788.372} C_VEL
LIN {X 0,Y 192.862,Z 416.46,A -85,B 0,C 180,E1 -21792.629,E2 -21792.629} C_VEL
LIN {X 0,Y 192.767,Z 416.463,A -85,B 0,C 180,E1 -21796.958,E2 -21796.958} C_VEL
LIN {X 0,Y 192.645,Z 416.462,A -85,B 0,C 180,E1 -21801.396,E2 -21801.396} C_VEL
LIN {X 0,Y 192.674,Z 416.481,A -85,B 0,C 180,E1 -21804.223,E2 -21804.223} C_VEL
LIN {X 0,Y 192.653,Z 416.484,A -85,B 0,C 180,E1 -21808.887,E2 -21808.887} C_VEL
LIN {X 0,Y 192.605,Z 416.465,A -85,B 0,C 180,E1 -21813.184,E2 -21813.184} C_VEL
LIN {X 0,Y 192.56,Z 416.498,A -85,B 0,C 180,E1 -21818.35,E2 -21818.35} C_VEL
LIN {X 0,Y 192.499,Z 416.486,A -85,B 0,C 180,E1 -21823.094,E2 -21823.094} C_VEL
LIN {X 0,Y 192.5,Z 416.502,A -85,B 0,C 180,E1 -21826.902,E2 -21826.902} C_VEL
LIN {X 0,Y 192.558,Z 416.486,A -85,B 0,C 180,E1 -21831.646,E2 -21831.646} C_VEL
LIN {X 0,Y 192.606,Z 416.498,A -85,B 0,C 180,E1 -21836.812,E2 -21836.812} C_VEL
LIN {X 0,Y 192.671,Z 416.488,A -85,B 0,C 180,E1 -21841.689,E2 -21841.689} C_VEL
LIN {X 0,Y 192.712,Z 416.475,A -85,B 0,C 180,E1 -21846.345,E2 -21846.345} C_VEL
LIN {X 0,Y 192.737,Z 416.473,A -85,B 0,C 180,E1 -21851.454,E2 -21851.454} C_VEL
LIN {X 0,Y 192.727,Z 416.605,A -85,B 0,C 180,E1 -21856.433,E2 -21856.433} C_VEL
LIN {X 0,Y 193.782,Z 419.483,A -85,B 0,C 180,E1 -21856.837,E2 -21856.837} C_VEL
LIN {X 0,Y 197.668,Z 427.714,A -85,B 0,C 180,E1 -21858.224,E2 -21858.224} C_VEL
LIN {X 0,Y 200.742,Z 436.239,A -85,B 0,C 180,E1 -21859.665,E2 -21859.665} C_VEL
LIN {X 0,Y 203.272,Z 447.591,A -85,B 0,C 180,E1 -21861.607,E2 -21861.607} C_VEL
LIN {X 0,Y 205.291,Z 458.84,A -85,B 0,C 180,E1 -21863.843,E2 -21863.843} C_VEL
LIN {X 0,Y 205.969,Z 463.264,A -85,B 0,C 180,E1 -21864.816,E2 -21864.816} C_VEL
LIN {X 0,Y 203.366,Z 474.285,A -85,B 0,C 180,E1 -21867.024,E2 -21867.024} C_VEL
LIN {X 0,Y 200.707,Z 484.064,A -85,B 0,C 180,E1 -21869.495,E2 -21869.495} C_VEL
LIN {X 0,Y 198.028,Z 493.042,A -85,B 0,C 180,E1 -21872.392,E2 -21872.392} C_VEL
LIN {X 0,Y 195.593,Z 500.993,A -85,B 0,C 180,E1 -21875.667,E2 -21875.667} C_VEL
LIN {X 0,Y 194.041,Z 506.064,A -85,B 0,C 180,E1 -21878.326,E2 -21878.326} C_VEL
LIN {X 0,Y 192.607,Z 510.833,A -85,B 0,C 180,E1 -21881.466,E2 -21881.466} C_VEL
LIN {X 0,Y 191.473,Z 514.724,A -85,B 0,C 180,E1 -21884.884,E2 -21884.884} C_VEL
LIN {X 0,Y 190.871,Z 516.595,A -85,B 0,C 180,E1 -21887.127,E2 -21887.127} C_VEL
LIN {X 0,Y 190.514,Z 518.014,A -85,B 0,C 180,E1 -21889.386,E2 -21889.386} C_VEL
LIN {X 0,Y 190.334,Z 519.232,A -85,B 0,C 180,E1 -21892.615,E2 -21892.615} C_VEL
LIN {X 0,Y 190.593,Z 519.516,A -85,B 0,C 180,E1 -21896.258,E2 -21896.258} C_VEL
LIN {X 0,Y 191.017,Z 519.099,A -85,B 0,C 180,E1 -21898.569,E2 -21898.569} C_VEL
LIN {X 0,Y 192.27,Z 517.064,A -85,B 0,C 180,E1 -21902.784,E2 -21902.784} C_VEL
LIN {X 0,Y 193.425,Z 514.837,A -85,B 0,C 180,E1 -21905.54,E2 -21905.54} C_VEL
LIN {X 0,Y 195.438,Z 510.874,A -85,B 0,C 180,E1 -21908.993,E2 -21908.993} C_VEL
LIN {X 0,Y 197.954,Z 505.511,A -85,B 0,C 180,E1 -21912.414,E2 -21912.414} C_VEL
LIN {X 0,Y 201.05,Z 498.735,A -85,B 0,C 180,E1 -21915.643,E2 -21915.643} C_VEL
LIN {X 0,Y 204.158,Z 491.096,A -85,B 0,C 180,E1 -21918.473,E2 -21918.473} C_VEL
LIN {X 0,Y 207.636,Z 481.97,A -85,B 0,C 180,E1 -21921.116,E2 -21921.116} C_VEL
LIN {X 0,Y 211.126,Z 471.699,A -85,B 0,C 180,E1 -21923.417,E2 -21923.417} C_VEL
LIN {X 0,Y 211.282,Z 469.17,A -85,B 0,C 180,E1 -21924.039,E2 -21924.039} C_VEL
LIN {X 0,Y 210.176,Z 459.577,A -85,B 0,C 180,E1 -21926.515,E2 -21926.515} C_VEL
LIN {X 0,Y 207.97,Z 449.726,A -85,B 0,C 180,E1 -21928.979,E2 -21928.979} C_VEL
LIN {X 0,Y 204.845,Z 440.701,A -85,B 0,C 180,E1 -21931.294,E2 -21931.294} C_VEL
LIN {X 0,Y 200.826,Z 432.203,A -85,B 0,C 180,E1 -21933.64,E2 -21933.64} C_VEL
LIN {X 0,Y 198.507,Z 428.183,A -85,B 0,C 180,E1 -21934.859,E2 -21934.859} C_VEL
LIN {X 0,Y 196.405,Z 424.615,A -85,B 0,C 180,E1 -21935.966,E2 -21935.966} C_VEL
LIN {X 0,Y 193.74,Z 420.982,A -85,B 0,C 180,E1 -21937.26,E2 -21937.26} C_VEL
LIN {X 0,Y 193.118,Z 419.114,A -85,B 0,C 180,E1 -21937.676,E2 -21937.676} C_VEL
LIN {X 0,Y 193.016,Z 418.073,A -85,B 0,C 180,E1 -21941.193,E2 -21941.193} C_VEL
LIN {X 0,Y 192.86,Z 417.083,A -85,B 0,C 180,E1 -21945.221,E2 -21945.221} C_VEL
LIN {X 0,Y 192.965,Z 416.443,A -85,B 0,C 180,E1 -21949.508,E2 -21949.508} C_VEL
LIN {X 0,Y 193.046,Z 416.439,A -85,B 0,C 180,E1 -21951.627,E2 -21951.627} C_VEL
LIN {X 0,Y 193.249,Z 416.414,A -85,B 0,C 180,E1 -21957.916,E2 -21957.916} C_VEL
LIN {X 0,Y 193.43,Z 416.391,A -85,B 0,C 180,E1 -21960,E2 -21960} C_VEL
LIN {X 0,Y 192.979,Z 416.446,A -85,B 0,C 180,E1 -21964.177,E2 -21964.177} C_VEL
LIN {X 0,Y 193.046,Z 416.44,A -85,B 0,C 180,E1 -21968.374,E2 -21968.374} C_VEL
LIN {X 0,Y 192.838,Z 416.464,A -85,B 0,C 180,E1 -21972.631,E2 -21972.631} C_VEL
LIN {X 0,Y 192.885,Z 417.281,A -85,B 0,C 180,E1 -21976.947,E2 -21976.947} C_VEL
LIN {X 0,Y 193.054,Z 418.629,A -85,B 0,C 180,E1 -21981.349,E2 -21981.349} C_VEL
LIN {X 0,Y 193.275,Z 419.85,A -85,B 0,C 180,E1 -21984.635,E2 -21984.635} C_VEL
LIN {X 0,Y 193.602,Z 421.972,A -85,B 0,C 180,E1 -21989.408,E2 -21989.408} C_VEL
LIN {X 0,Y 193.949,Z 424.132,A -85,B 0,C 180,E1 -21993.556,E2 -21993.556} C_VEL
LIN {X 0,Y 194.398,Z 426.738,A -85,B 0,C 180,E1 -21997.923,E2 -21997.923} C_VEL
LIN {X 0,Y 194.714,Z 428.594,A -85,B 0,C 180,E1 -22000.722,E2 -22000.722} C_VEL
LIN {X 0,Y 195.491,Z 432.453,A -85,B 0,C 180,E1 -22006.072,E2 -22006.072} C_VEL
LIN {X 0,Y 196.741,Z 435.864,A -85,B 0,C 180,E1 -22006.794,E2 -22006.794} C_VEL
LIN {X 0,Y 198.7,Z 438.809,A -85,B 0,C 180,E1 -22007.692,E2 -22007.692} C_VEL
LIN {X 0,Y 200.675,Z 442.88,A -85,B 0,C 180,E1 -22008.691,E2 -22008.691} C_VEL
LIN {X 0,Y 203.07,Z 449.149,A -85,B 0,C 180,E1 -22010.068,E2 -22010.068} C_VEL
LIN {X 0,Y 205.076,Z 457.106,A -85,B 0,C 180,E1 -22011.622,E2 -22011.622} C_VEL
LIN {X 0,Y 206.761,Z 468.933,A -85,B 0,C 180,E1 -22013.878,E2 -22013.878} C_VEL
LIN {X 0,Y 207.297,Z 478.904,A -85,B 0,C 180,E1 -22015.879,E2 -22015.879} C_VEL
LIN {X 0,Y 206.961,Z 489.097,A -85,B 0,C 180,E1 -22018.098,E2 -22018.098} C_VEL
LIN {X 0,Y 205.799,Z 498.356,A -85,B 0,C 180,E1 -22020.324,E2 -22020.324} C_VEL
LIN {X 0,Y 204.599,Z 503.981,A -85,B 0,C 180,E1 -22021.82,E2 -22021.82} C_VEL
LIN {X 0,Y 200.863,Z 513.589,A -85,B 0,C 180,E1 -22024.625,E2 -22024.625} C_VEL
LIN {X 0,Y 197.957,Z 520.905,A -85,B 0,C 180,E1 -22027.38,E2 -22027.38} C_VEL
LIN {X 0,Y 195.699,Z 526.609,A -85,B 0,C 180,E1 -22030.057,E2 -22030.057} C_VEL
LIN {X 0,Y 193.571,Z 531.804,A -85,B 0,C 180,E1 -22033.119,E2 -22033.119} C_VEL
LIN {X 0,Y 191.758,Z 536.55,A -85,B 0,C 180,E1 -22036.872,E2 -22036.872} C_VEL
LIN {X 0,Y 191.028,Z 538.95,A -85,B 0,C 180,E1 -22039.404,E2 -22039.404} C_VEL
LIN {X 0,Y 190.63,Z 540.453,A -85,B 0,C 180,E1 -22041.524,E2 -22041.524} C_VEL
LIN {X 0,Y 190.384,Z 542.256,A -85,B 0,C 180,E1 -22045.77,E2 -22045.77} C_VEL
LIN {X 0,Y 190.383,Z 542.271,A -85,B 0,C 180,E1 -22045.868,E2 -22045.868} C_VEL
LIN {X 0,Y 190.063,Z 542.465,A -85,B 0,C 180,E1 -22047.051,E2 -22047.051} C_VEL
LIN {X 0,Y 188.734,Z 542.472,A -85,B 0,C 180,E1 -22048.801,E2 -22048.801} C_VEL
LIN {X 0,Y 184.496,Z 541.287,A -85,B 0,C 180,E1 -22052.893,E2 -22052.893} C_VEL
LIN {X 0,Y 183.473,Z 540.316,A -85,B 0,C 180,E1 -22054.713,E2 -22054.713} C_VEL
LIN {X 0,Y 183.391,Z 539.927,A -85,B 0,C 180,E1 -22055.327,E2 -22055.327} C_VEL
LIN {X 0,Y 183.661,Z 537.225,A -85,B 0,C 180,E1 -22058.809,E2 -22058.809} C_VEL
LIN {X 0,Y 184.331,Z 533.594,A -85,B 0,C 180,E1 -22062.109,E2 -22062.109} C_VEL
LIN {X 0,Y 185.504,Z 528.834,A -85,B 0,C 180,E1 -22065.383,E2 -22065.383} C_VEL
LIN {X 0,Y 187.299,Z 522.814,A -85,B 0,C 180,E1 -22068.603,E2 -22068.603} C_VEL
LIN {X 0,Y 189.219,Z 516.679,A -85,B 0,C 180,E1 -22071.235,E2 -22071.235} C_VEL
LIN {X 0,Y 191.857,Z 507.646,A -85,B 0,C 180,E1 -22074.341,E2 -22074.341} C_VEL
LIN {X 0,Y 194.539,Z 498.363,A -85,B 0,C 180,E1 -22076.849,E2 -22076.849} C_VEL
LIN {X 0,Y 195.133,Z 488.075,A -85,B 0,C 180,E1 -22079.291,E2 -22079.291} C_VEL
LIN {X 0,Y 195.01,Z 477.127,A -85,B 0,C 180,E1 -22081.509,E2 -22081.509} C_VEL
LIN {X 0,Y 194.133,Z 464.86,A -85,B 0,C 180,E1 -22083.628,E2 -22083.628} C_VEL
LIN {X 0,Y 192.273,Z 451.977,A -85,B 0,C 180,E1 -22085.527,E2 -22085.527} C_VEL
LIN {X 0,Y 189.424,Z 439.084,A -85,B 0,C 180,E1 -22087.179,E2 -22087.179} C_VEL
LIN {X 0,Y 188.343,Z 434.796,A -85,B 0,C 180,E1 -22087.678,E2 -22087.678} C_VEL
LIN {X 0,Y 188.298,Z 432.264,A -85,B 0,C 180,E1 -22090.481,E2 -22090.481} C_VEL
LIN {X 0,Y 187.551,Z 428.069,A -85,B 0,C 180,E1 -22095.401,E2 -22095.401} C_VEL
LIN {X 0,Y 186.742,Z 424.269,A -85,B 0,C 180,E1 -22100.223,E2 -22100.223} C_VEL
LIN {X 0,Y 186.067,Z 420.439,A -85,B 0,C 180,E1 -22105.488,E2 -22105.488} C_VEL
LIN {X 0,Y 185.615,Z 417.369,A -85,B 0,C 180,E1 -22110.201,E2 -22110.201} C_VEL
LIN {X 0,Y 185.597,Z 417.367,A -85,B 0,C 180,E1 -22115.384,E2 -22115.384} C_VEL
LIN {X 0,Y 185.685,Z 417.36,A -85,B 0,C 180,E1 -22121.134,E2 -22121.134} C_VEL
LIN {X 0,Y 185.704,Z 417.36,A -85,B 0,C 180,E1 -22124.638,E2 -22124.638} C_VEL
LIN {X 0,Y 185.899,Z 417.332,A -85,B 0,C 180,E1 -22129.418,E2 -22129.418} C_VEL
LIN {X 0,Y 185.956,Z 417.323,A -85,B 0,C 180,E1 -22133.49,E2 -22133.49} C_VEL
LIN {X 0,Y 186.215,Z 417.29,A -85,B 0,C 180,E1 -22137.837,E2 -22137.837} C_VEL
LIN {X 0,Y 186.414,Z 417.265,A -85,B 0,C 180,E1 -22140,E2 -22140} C_VEL
LIN {X 0,Y 185.931,Z 417.308,A -85,B 0,C 180,E1 -22144.335,E2 -22144.335} C_VEL
LIN {X 0,Y 186.019,Z 417.289,A -85,B 0,C 180,E1 -22148.692,E2 -22148.692} C_VEL
LIN {X 0,Y 185.774,Z 417.343,A -85,B 0,C 180,E1 -22153.12,E2 -22153.12} C_VEL
LIN {X 0,Y 185.7,Z 417.336,A -85,B 0,C 180,E1 -22157.624,E2 -22157.624} C_VEL
LIN {X 0,Y 185.606,Z 417.344,A -85,B 0,C 180,E1 -22162.25,E2 -22162.25} C_VEL
LIN {X 0,Y 185.57,Z 417.369,A -85,B 0,C 180,E1 -22167.031,E2 -22167.031} C_VEL
LIN {X 0,Y 185.587,Z 417.358,A -85,B 0,C 180,E1 -22169.492,E2 -22169.492} C_VEL
LIN {X 0,Y 185.507,Z 417.36,A -85,B 0,C 180,E1 -22174.63,E2 -22174.63} C_VEL
LIN {X 0,Y 185.514,Z 417.375,A -85,B 0,C 180,E1 -22177.311,E2 -22177.311} C_VEL
LIN {X 0,Y 185.48,Z 417.376,A -85,B 0,C 180,E1 -22180.723,E2 -22180.723} C_VEL
LIN {X 0,Y 185.486,Z 417.373,A -85,B 0,C 180,E1 -22186.046,E2 -22186.046} C_VEL
LIN {X 0,Y 185.476,Z 417.378,A -85,B 0,C 180,E1 -22189.893,E2 -22189.893} C_VEL
LIN {X 0,Y 185.513,Z 417.361,A -85,B 0,C 180,E1 -22192.709,E2 -22192.709} C_VEL
LIN {X 0,Y 185.553,Z 417.372,A -85,B 0,C 180,E1 -22197.973,E2 -22197.973} C_VEL
LIN {X 0,Y 185.588,Z 417.36,A -85,B 0,C 180,E1 -22200.573,E2 -22200.573} C_VEL
LIN {X 0,Y 185.594,Z 417.363,A -85,B 0,C 180,E1 -22205.379,E2 -22205.379} C_VEL
LIN {X 0,Y 185.613,Z 417.362,A -85,B 0,C 180,E1 -22210.072,E2 -22210.072} C_VEL
LIN {X 0,Y 185.689,Z 417.354,A -85,B 0,C 180,E1 -22212.371,E2 -22212.371} C_VEL
LIN {X 0,Y 185.662,Z 417.359,A -85,B 0,C 180,E1 -22215.073,E2 -22215.073} C_VEL
LIN {X 0,Y 186.742,Z 420.332,A -85,B 0,C 180,E1 -22215.521,E2 -22215.521} C_VEL
LIN {X 0,Y 189.876,Z 426.378,A -85,B 0,C 180,E1 -22216.661,E2 -22216.661} C_VEL
LIN {X 0,Y 193.699,Z 436.012,A -85,B 0,C 180,E1 -22218.419,E2 -22218.419} C_VEL
LIN {X 0,Y 195.895,Z 444.366,A -85,B 0,C 180,E1 -22219.923,E2 -22219.923} C_VEL
LIN {X 0,Y 197.956,Z 455.393,A -85,B 0,C 180,E1 -22222.089,E2 -22222.089} C_VEL
LIN {X 0,Y 199.244,Z 465.272,A -85,B 0,C 180,E1 -22224.29,E2 -22224.29} C_VEL
LIN {X 0,Y 196.667,Z 475.388,A -85,B 0,C 180,E1 -22226.411,E2 -22226.411} C_VEL
LIN {X 0,Y 193.877,Z 485.022,A -85,B 0,C 180,E1 -22228.957,E2 -22228.957} C_VEL
LIN {X 0,Y 190.984,Z 494.317,A -85,B 0,C 180,E1 -22232.105,E2 -22232.105} C_VEL
LIN {X 0,Y 188.618,Z 501.767,A -85,B 0,C 180,E1 -22235.341,E2 -22235.341} C_VEL
LIN {X 0,Y 186.721,Z 507.671,A -85,B 0,C 180,E1 -22238.655,E2 -22238.655} C_VEL
LIN {X 0,Y 185.284,Z 512.305,A -85,B 0,C 180,E1 -22242.037,E2 -22242.037} C_VEL
LIN {X 0,Y 184.186,Z 515.806,A -85,B 0,C 180,E1 -22245.487,E2 -22245.487} C_VEL
LIN {X 0,Y 183.659,Z 517.554,A -85,B 0,C 180,E1 -22247.822,E2 -22247.822} C_VEL
LIN {X 0,Y 183.334,Z 518.828,A -85,B 0,C 180,E1 -22250.177,E2 -22250.177} C_VEL
LIN {X 0,Y 183.253,Z 519.733,A -85,B 0,C 180,E1 -22253.011,E2 -22253.011} C_VEL
LIN {X 0,Y 183.371,Z 519.985,A -85,B 0,C 180,E1 -22254.93,E2 -22254.93} C_VEL
LIN {X 0,Y 183.912,Z 519.65,A -85,B 0,C 180,E1 -22258.487,E2 -22258.487} C_VEL
LIN {X 0,Y 184.922,Z 518.23,A -85,B 0,C 180,E1 -22262.14,E2 -22262.14} C_VEL
LIN {X 0,Y 186.397,Z 515.673,A -85,B 0,C 180,E1 -22265.756,E2 -22265.756} C_VEL
LIN {X 0,Y 188.486,Z 511.861,A -85,B 0,C 180,E1 -22269.33,E2 -22269.33} C_VEL
LIN {X 0,Y 191.38,Z 506.092,A -85,B 0,C 180,E1 -22273.197,E2 -22273.197} C_VEL
LIN {X 0,Y 194.416,Z 499.888,A -85,B 0,C 180,E1 -22276.295,E2 -22276.295} C_VEL
LIN {X 0,Y 197.53,Z 492.703,A -85,B 0,C 180,E1 -22279.111,E2 -22279.111} C_VEL
LIN {X 0,Y 201.13,Z 483.815,A -85,B 0,C 180,E1 -22281.825,E2 -22281.825} C_VEL
LIN {X 0,Y 204.37,Z 475.005,A -85,B 0,C 180,E1 -22283.956,E2 -22283.956} C_VEL
LIN {X 0,Y 205.055,Z 473.091,A -85,B 0,C 180,E1 -22284.363,E2 -22284.363} C_VEL
LIN {X 0,Y 204.789,Z 466.148,A -85,B 0,C 180,E1 -22286.262,E2 -22286.262} C_VEL
LIN {X 0,Y 203.3,Z 456.92,A -85,B 0,C 180,E1 -22288.766,E2 -22288.766} C_VEL
LIN {X 0,Y 200.849,Z 447.833,A -85,B 0,C 180,E1 -22291.241,E2 -22291.241} C_VEL
LIN {X 0,Y 197.614,Z 439.66,A -85,B 0,C 180,E1 -22293.605,E2 -22293.605} C_VEL
LIN {X 0,Y 194.412,Z 433.472,A -85,B 0,C 180,E1 -22295.586,E2 -22295.586} C_VEL
LIN {X 0,Y 191.821,Z 429.132,A -85,B 0,C 180,E1 -22297.09,E2 -22297.09} C_VEL
LIN {X 0,Y 189.806,Z 425.815,A -85,B 0,C 180,E1 -22298.268,E2 -22298.268} C_VEL
LIN {X 0,Y 189.122,Z 424.762,A -85,B 0,C 180,E1 -22298.657,E2 -22298.657} C_VEL
LIN {X 0,Y 186.895,Z 422.115,A -85,B 0,C 180,E1 -22299.864,E2 -22299.864} C_VEL
LIN {X 0,Y 186.082,Z 419.805,A -85,B 0,C 180,E1 -22300.54,E2 -22300.54} C_VEL
LIN {X 0,Y 185.932,Z 418.821,A -85,B 0,C 180,E1 -22304.657,E2 -22304.657} C_VEL
LIN {X 0,Y 185.983,Z 417.901,A -85,B 0,C 180,E1 -22309.236,E2 -22309.236} C_VEL
LIN {X 0,Y 186.031,Z 417.562,A -85,B 0,C 180,E1 -22311.309,E2 -22311.309} C_VEL
LIN {X 0,Y 185.911,Z 417.326,A -85,B 0,C 180,E1 -22315.664,E2 -22315.664} C_VEL
LIN {X 0,Y 186.393,Z 417.267,A -85,B 0,C 180,E1 -22320,E2 -22320} C_VEL
LIN {X 0,Y 185.925,Z 417.324,A -85,B 0,C 180,E1 -22324.336,E2 -22324.336} C_VEL
LIN {X 0,Y 185.993,Z 417.396,A -85,B 0,C 180,E1 -22328.694,E2 -22328.694} C_VEL
LIN {X 0,Y 185.901,Z 418.167,A -85,B 0,C 180,E1 -22333.111,E2 -22333.111} C_VEL
LIN {X 0,Y 186.024,Z 419.223,A -85,B 0,C 180,E1 -22337.592,E2 -22337.592} C_VEL
LIN {X 0,Y 186.218,Z 420.65,A -85,B 0,C 180,E1 -22342.173,E2 -22342.173} C_VEL
LIN {X 0,Y 186.411,Z 421.778,A -85,B 0,C 180,E1 -22345.211,E2 -22345.211} C_VEL
LIN {X 0,Y 186.717,Z 423.915,A -85,B 0,C 180,E1 -22350.046,E2 -22350.046} C_VEL
LIN {X 0,Y 187.064,Z 426.128,A -85,B 0,C 180,E1 -22354.302,E2 -22354.302} C_VEL
LIN {X 0,Y 187.484,Z 428.324,A -85,B 0,C 180,E1 -22358.083,E2 -22358.083} C_VEL
LIN {X 0,Y 188.112,Z 431.768,A -85,B 0,C 180,E1 -22363.308,E2 -22363.308} C_VEL
LIN {X 0,Y 189.241,Z 434.87,A -85,B 0,C 180,E1 -22364.034,E2 -22364.034} C_VEL
LIN {X 0,Y 191.689,Z 438.436,A -85,B 0,C 180,E1 -22365.287,E2 -22365.287} C_VEL
LIN {X 0,Y 193.673,Z 442.464,A -85,B 0,C 180,E1 -22366.418,E2 -22366.418} C_VEL
LIN {X 0,Y 194.719,Z 444.5,A -85,B 0,C 180,E1 -22366.997,E2 -22366.997} C_VEL
LIN {X 0,Y 197.15,Z 450.095,A -85,B 0,C 180,E1 -22368.47,E2 -22368.47} C_VEL
LIN {X 0,Y 198.933,Z 456.339,A -85,B 0,C 180,E1 -22369.857,E2 -22369.857} C_VEL
LIN {X 0,Y 200.637,Z 467.347,A -85,B 0,C 180,E1 -22372.125,E2 -22372.125} C_VEL
LIN {X 0,Y 201.224,Z 478.519,A -85,B 0,C 180,E1 -22374.483,E2 -22374.483} C_VEL
LIN {X 0,Y 200.802,Z 489.376,A -85,B 0,C 180,E1 -22376.97,E2 -22376.97} C_VEL
LIN {X 0,Y 199.537,Z 498.561,A -85,B 0,C 180,E1 -22379.294,E2 -22379.294} C_VEL
LIN {X 0,Y 198.321,Z 504.106,A -85,B 0,C 180,E1 -22380.844,E2 -22380.844} C_VEL
LIN {X 0,Y 194.447,Z 513.578,A -85,B 0,C 180,E1 -22383.725,E2 -22383.725} C_VEL
LIN {X 0,Y 191.202,Z 521.272,A -85,B 0,C 180,E1 -22386.77,E2 -22386.77} C_VEL
LIN {X 0,Y 189.034,Z 526.453,A -85,B 0,C 180,E1 -22389.322,E2 -22389.322} C_VEL
LIN {X 0,Y 186.76,Z 531.586,A -85,B 0,C 180,E1 -22392.484,E2 -22392.484} C_VEL
LIN {X 0,Y 185.036,Z 535.611,A -85,B 0,C 180,E1 -22395.712,E2 -22395.712} C_VEL
LIN {X 0,Y 184.032,Z 538.634,A -85,B 0,C 180,E1 -22398.997,E2 -22398.997} C_VEL
LIN {X 0,Y 183.358,Z 541.169,A -85,B 0,C 180,E1 -22403.401,E2 -22403.401} C_VEL
LIN {X 0,Y 183.303,Z 541.89,A -85,B 0,C 180,E1 -22405.867,E2 -22405.867} C_VEL
LIN {X 0,Y 183.392,Z 542.151,A -85,B 0,C 180,E1 -22407.808,E2 -22407.808} C_VEL
LIN {X 0,Y 183.54,Z 542.008,A -85,B 0,C 180,E1 -22410.004,E2 -22410.004} C_VEL
LIN {X 0,Y 183.437,Z 541.439,A -85,B 0,C 180,E1 -22412.2,E2 -22412.2} C_VEL
LIN {X 0,Y 183.391,Z 539.927,A -85,B 0,C 180,E1 -22415.327,E2 -22415.327} C_VEL
LIN {X 0,Y 182.786,Z 538.649,A -85,B 0,C 180,E1 -22417.118,E2 -22417.118} C_VEL
LIN {X 0,Y 180.298,Z 535.933,A -85,B 0,C 180,E1 -22420.025,E2 -22420.025} C_VEL
LIN {X 0,Y 178.421,Z 533.25,A -85,B 0,C 180,E1 -22422.354,E2 -22422.354} C_VEL
LIN {X 0,Y 177.935,Z 530.949,A -85,B 0,C 180,E1 -22424.111,E2 -22424.111} C_VEL
LIN {X 0,Y 178.063,Z 530.115,A -85,B 0,C 180,E1 -22424.691,E2 -22424.691} C_VEL
LIN {X 0,Y 179.918,Z 524.244,A -85,B 0,C 180,E1 -22428.214,E2 -22428.214} C_VEL
LIN {X 0,Y 182.167,Z 517.193,A -85,B 0,C 180,E1 -22431.505,E2 -22431.505} C_VEL
LIN {X 0,Y 184.273,Z 510.137,A -85,B 0,C 180,E1 -22434.149,E2 -22434.149} C_VEL
LIN {X 0,Y 187.042,Z 501.263,A -85,B 0,C 180,E1 -22436.805,E2 -22436.805} C_VEL
LIN {X 0,Y 187.892,Z 497.207,A -85,B 0,C 180,E1 -22437.88,E2 -22437.88} C_VEL
LIN {X 0,Y 188.479,Z 486.617,A -85,B 0,C 180,E1 -22440.459,E2 -22440.459} C_VEL
LIN {X 0,Y 188.287,Z 475.886,A -85,B 0,C 180,E1 -22442.706,E2 -22442.706} C_VEL
LIN {X 0,Y 187.518,Z 464.693,A -85,B 0,C 180,E1 -22444.715,E2 -22444.715} C_VEL
LIN {X 0,Y 185.969,Z 453.342,A -85,B 0,C 180,E1 -22446.493,E2 -22446.493} C_VEL
LIN {X 0,Y 183.331,Z 440.812,A -85,B 0,C 180,E1 -22448.22,E2 -22448.22} C_VEL
LIN {X 0,Y 181.401,Z 434.906,A -85,B 0,C 180,E1 -22449.04,E2 -22449.04} C_VEL
LIN {X 0,Y 181.323,Z 434.263,A -85,B 0,C 180,E1 -22449.177,E2 -22449.177} C_VEL
LIN {X 0,Y 180.943,Z 431.499,A -85,B 0,C 180,E1 -22452.44,E2 -22452.44} C_VEL
LIN {X 0,Y 180.505,Z 429.049,A -85,B 0,C 180,E1 -22455.505,E2 -22455.505} C_VEL
LIN {X 0,Y 179.818,Z 425.728,A -85,B 0,C 180,E1 -22459.843,E2 -22459.843} C_VEL
LIN {X 0,Y 179.108,Z 421.767,A -85,B 0,C 180,E1 -22465.495,E2 -22465.495} C_VEL
LIN {X 0,Y 178.544,Z 418.275,A -85,B 0,C 180,E1 -22470.982,E2 -22470.982} C_VEL
LIN {X 0,Y 178.535,Z 418.247,A -85,B 0,C 180,E1 -22474.884,E2 -22474.884} C_VEL
LIN {X 0,Y 178.634,Z 418.24,A -85,B 0,C 180,E1 -22480.785,E2 -22480.785} C_VEL
LIN {X 0,Y 178.667,Z 418.237,A -85,B 0,C 180,E1 -22486.348,E2 -22486.348} C_VEL
LIN {X 0,Y 178.921,Z 418.201,A -85,B 0,C 180,E1 -22490.96,E2 -22490.96} C_VEL
LIN {X 0,Y 179.16,Z 418.169,A -85,B 0,C 180,E1 -22497.752,E2 -22497.752} C_VEL
LIN {X 0,Y 179.377,Z 418.142,A -85,B 0,C 180,E1 -22500,E2 -22500} C_VEL
LIN {X 0,Y 178.879,Z 418.185,A -85,B 0,C 180,E1 -22504.507,E2 -22504.507} C_VEL
LIN {X 0,Y 178.97,Z 418.17,A -85,B 0,C 180,E1 -22509.037,E2 -22509.037} C_VEL
LIN {X 0,Y 178.696,Z 418.227,A -85,B 0,C 180,E1 -22513.649,E2 -22513.649} C_VEL
LIN {X 0,Y 178.66,Z 418.207,A -85,B 0,C 180,E1 -22518.342,E2 -22518.342} C_VEL
LIN {X 0,Y 178.52,Z 418.234,A -85,B 0,C 180,E1 -22523.184,E2 -22523.184} C_VEL
LIN {X 0,Y 178.495,Z 418.247,A -85,B 0,C 180,E1 -22528.195,E2 -22528.195} C_VEL
LIN {X 0,Y 178.486,Z 418.231,A -85,B 0,C 180,E1 -22530.789,E2 -22530.789} C_VEL
LIN {X 0,Y 178.493,Z 418.228,A -85,B 0,C 180,E1 -22534.217,E2 -22534.217} C_VEL
LIN {X 0,Y 178.404,Z 418.263,A -85,B 0,C 180,E1 -22539.072,E2 -22539.072} C_VEL
LIN {X 0,Y 178.407,Z 418.247,A -85,B 0,C 180,E1 -22542.042,E2 -22542.042} C_VEL
LIN {X 0,Y 178.409,Z 418.245,A -85,B 0,C 180,E1 -22545.159,E2 -22545.159} C_VEL
LIN {X 0,Y 178.411,Z 418.261,A -85,B 0,C 180,E1 -22548.456,E2 -22548.456} C_VEL
LIN {X 0,Y 178.429,Z 418.248,A -85,B 0,C 180,E1 -22553.78,E2 -22553.78} C_VEL
LIN {X 0,Y 178.494,Z 418.255,A -85,B 0,C 180,E1 -22556.544,E2 -22556.544} C_VEL
LIN {X 0,Y 178.529,Z 418.237,A -85,B 0,C 180,E1 -22560.003,E2 -22560.003} C_VEL
LIN {X 0,Y 178.54,Z 418.244,A -85,B 0,C 180,E1 -22564.872,E2 -22564.872} C_VEL
LIN {X 0,Y 178.628,Z 418.229,A -85,B 0,C 180,E1 -22570.78,E2 -22570.78} C_VEL
LIN {X 0,Y 178.615,Z 418.37,A -85,B 0,C 180,E1 -22573.641,E2 -22573.641} C_VEL
LIN {X 0,Y 179.687,Z 421.229,A -85,B 0,C 180,E1 -22574.106,E2 -22574.106} C_VEL
LIN {X 0,Y 180.901,Z 423.227,A -85,B 0,C 180,E1 -22574.535,E2 -22574.535} C_VEL
LIN {X 0,Y 185.119,Z 431.928,A -85,B 0,C 180,E1 -22576.295,E2 -22576.295} C_VEL
LIN {X 0,Y 188.328,Z 440.976,A -85,B 0,C 180,E1 -22578.084,E2 -22578.084} C_VEL
LIN {X 0,Y 189.995,Z 448.584,A -85,B 0,C 180,E1 -22579.551,E2 -22579.551} C_VEL
LIN {X 0,Y 191.846,Z 459.705,A -85,B 0,C 180,E1 -22581.944,E2 -22581.944} C_VEL
LIN {X 0,Y 192.614,Z 465.407,A -85,B 0,C 180,E1 -22583.311,E2 -22583.311} C_VEL
LIN {X 0,Y 192.2,Z 468.323,A -85,B 0,C 180,E1 -22583.93,E2 -22583.93} C_VEL
LIN {X 0,Y 189.351,Z 478.518,A -85,B 0,C 180,E1 -22586.272,E2 -22586.272} C_VEL
LIN {X 0,Y 186.538,Z 487.658,A -85,B 0,C 180,E1 -22588.916,E2 -22588.916} C_VEL
LIN {X 0,Y 184.106,Z 495.174,A -85,B 0,C 180,E1 -22591.636,E2 -22591.636} C_VEL
LIN {X 0,Y 181.621,Z 502.527,A -85,B 0,C 180,E1 -22594.99,E2 -22594.99} C_VEL
LIN {X 0,Y 179.955,Z 507.51,A -85,B 0,C 180,E1 -22597.852,E2 -22597.852} C_VEL
LIN {X 0,Y 178.404,Z 512.279,A -85,B 0,C 180,E1 -22601.355,E2 -22601.355} C_VEL
LIN {X 0,Y 177.223,Z 515.902,A -85,B 0,C 180,E1 -22604.933,E2 -22604.933} C_VEL
LIN {X 0,Y 176.428,Z 518.452,A -85,B 0,C 180,E1 -22608.578,E2 -22608.578} C_VEL
LIN {X 0,Y 176.185,Z 519.563,A -85,B 0,C 180,E1 -22611.034,E2 -22611.034} C_VEL
LIN {X 0,Y 176.194,Z 520.245,A -85,B 0,C 180,E1 -22613.503,E2 -22613.503} C_VEL
LIN {X 0,Y 176.385,Z 520.43,A -85,B 0,C 180,E1 -22615.989,E2 -22615.989} C_VEL
LIN {X 0,Y 176.947,Z 520.05,A -85,B 0,C 180,E1 -22619.097,E2 -22619.097} C_VEL
LIN {X 0,Y 178.31,Z 518.198,A -85,B 0,C 180,E1 -22623.485,E2 -22623.485} C_VEL
LIN {X 0,Y 180.024,Z 515.384,A -85,B 0,C 180,E1 -22627.23,E2 -22627.23} C_VEL
LIN {X 0,Y 182.378,Z 511.308,A -85,B 0,C 180,E1 -22630.921,E2 -22630.921} C_VEL
LIN {X 0,Y 185.341,Z 505.75,A -85,B 0,C 180,E1 -22634.581,E2 -22634.581} C_VEL
LIN {X 0,Y 188.942,Z 498.611,A -85,B 0,C 180,E1 -22638.06,E2 -22638.06} C_VEL
LIN {X 0,Y 192.257,Z 491.314,A -85,B 0,C 180,E1 -22640.837,E2 -22640.837} C_VEL
LIN {X 0,Y 196.295,Z 481.749,A -85,B 0,C 180,E1 -22643.657,E2 -22643.657} C_VEL
LIN {X 0,Y 198.852,Z 474.979,A -85,B 0,C 180,E1 -22645.257,E2 -22645.257} C_VEL
LIN {X 0,Y 198.8,Z 468.735,A -85,B 0,C 180,E1 -22647.075,E2 -22647.075} C_VEL
LIN {X 0,Y 197.676,Z 460.221,A -85,B 0,C 180,E1 -22649.56,E2 -22649.56} C_VEL
LIN {X 0,Y 195.515,Z 451.45,A -85,B 0,C 180,E1 -22652.141,E2 -22652.141} C_VEL
LIN {X 0,Y 192.59,Z 443.57,A -85,B 0,C 180,E1 -22654.61,E2 -22654.61} C_VEL
LIN {X 0,Y 190.585,Z 439.265,A -85,B 0,C 180,E1 -22656.069,E2 -22656.069} C_VEL
LIN {X 0,Y 187.773,Z 434.374,A -85,B 0,C 180,E1 -22657.921,E2 -22657.921} C_VEL
LIN {X 0,Y 185.407,Z 430.358,A -85,B 0,C 180,E1 -22659.501,E2 -22659.501} C_VEL
LIN {X 0,Y 183.203,Z 427.127,A -85,B 0,C 180,E1 -22660.916,E2 -22660.916} C_VEL
LIN {X 0,Y 182.482,Z 425.711,A -85,B 0,C 180,E1 -22661.43,E2 -22661.43} C_VEL
LIN {X 0,Y 179.999,Z 423.039,A -85,B 0,C 180,E1 -22662.972,E2 -22662.972} C_VEL
LIN {X 0,Y 179.012,Z 420.598,A -85,B 0,C 180,E1 -22663.829,E2 -22663.829} C_VEL
LIN {X 0,Y 179.044,Z 419.634,A -85,B 0,C 180,E1 -22668.881,E2 -22668.881} C_VEL
LIN {X 0,Y 179.12,Z 419.289,A -85,B 0,C 180,E1 -22670.971,E2 -22670.971} C_VEL
LIN {X 0,Y 179.226,Z 418.679,A -85,B 0,C 180,E1 -22677.753,E2 -22677.753} C_VEL
LIN {X 0,Y 179.412,Z 418.578,A -85,B 0,C 180,E1 -22680,E2 -22680} C_VEL
LIN {X 0,Y 178.976,Z 418.816,A -85,B 0,C 180,E1 -22684.505,E2 -22684.505} C_VEL
LIN {X 0,Y 179.109,Z 419.226,A -85,B 0,C 180,E1 -22689.03,E2 -22689.03} C_VEL
LIN {X 0,Y 179.028,Z 420.046,A -85,B 0,C 180,E1 -22693.624,E2 -22693.624} C_VEL
LIN {X 0,Y 179.183,Z 421.166,A -85,B 0,C 180,E1 -22698.287,E2 -22698.287} C_VEL
LIN {X 0,Y 179.373,Z 422.675,A -85,B 0,C 180,E1 -22703.067,E2 -22703.067} C_VEL
LIN {X 0,Y 179.627,Z 424.63,A -85,B 0,C 180,E1 -22708.003,E2 -22708.003} C_VEL
LIN {X 0,Y 179.846,Z 425.877,A -85,B 0,C 180,E1 -22710.726,E2 -22710.726} C_VEL
LIN {X 0,Y 180.257,Z 428.5,A -85,B 0,C 180,E1 -22715.791,E2 -22715.791} C_VEL
LIN {X 0,Y 180.696,Z 431.017,A -85,B 0,C 180,E1 -22719.987,E2 -22719.987} C_VEL
LIN {X 0,Y 181.91,Z 434.219,A -85,B 0,C 180,E1 -22720.88,E2 -22720.88} C_VEL
LIN {X 0,Y 184.529,Z 437.672,A -85,B 0,C 180,E1 -22722.411,E2 -22722.411} C_VEL
LIN {X 0,Y 186.395,Z 441.696,A -85,B 0,C 180,E1 -22723.669,E2 -22723.669} C_VEL
LIN {X 0,Y 187.771,Z 443.883,A -85,B 0,C 180,E1 -22724.478,E2 -22724.478} C_VEL
LIN {X 0,Y 190.573,Z 449.891,A -85,B 0,C 180,E1 -22726.305,E2 -22726.305} C_VEL
LIN {X 0,Y 192.491,Z 454.716,A -85,B 0,C 180,E1 -22727.677,E2 -22727.677} C_VEL
LIN {X 0,Y 194.141,Z 462.475,A -85,B 0,C 180,E1 -22729.483,E2 -22729.483} C_VEL
LIN {X 0,Y 195.135,Z 472.336,A -85,B 0,C 180,E1 -22731.668,E2 -22731.668} C_VEL
LIN {X 0,Y 195.202,Z 482.592,A -85,B 0,C 180,E1 -22734.026,E2 -22734.026} C_VEL
LIN {X 0,Y 194.344,Z 492.873,A -85,B 0,C 180,E1 -22736.589,E2 -22736.589} C_VEL
LIN {X 0,Y 192.53,Z 502.519,A -85,B 0,C 180,E1 -22739.272,E2 -22739.272} C_VEL
LIN {X 0,Y 190.8,Z 507.607,A -85,B 0,C 180,E1 -22740.792,E2 -22740.792} C_VEL
LIN {X 0,Y 186.899,Z 516.311,A -85,B 0,C 180,E1 -22743.784,E2 -22743.784} C_VEL
LIN {X 0,Y 184.109,Z 522.654,A -85,B 0,C 180,E1 -22746.593,E2 -22746.593} C_VEL
LIN {X 0,Y 181.474,Z 528.134,A -85,B 0,C 180,E1 -22749.607,E2 -22749.607} C_VEL
LIN {X 0,Y 179.296,Z 532.825,A -85,B 0,C 180,E1 -22752.908,E2 -22752.908} C_VEL
LIN {X 0,Y 177.71,Z 536.441,A -85,B 0,C 180,E1 -22756.278,E2 -22756.278} C_VEL
LIN {X 0,Y 177.022,Z 538.311,A -85,B 0,C 180,E1 -22758.555,E2 -22758.555} C_VEL
LIN {X 0,Y 176.299,Z 540.795,A -85,B 0,C 180,E1 -22763.136,E2 -22763.136} C_VEL
LIN {X 0,Y 176.226,Z 541.492,A -85,B 0,C 180,E1 -22765.575,E2 -22765.575} C_VEL
LIN {X 0,Y 176.308,Z 541.713,A -85,B 0,C 180,E1 -22767.72,E2 -22767.72} C_VEL
LIN {X 0,Y 176.474,Z 541.539,A -85,B 0,C 180,E1 -22770.004,E2 -22770.004} C_VEL
LIN {X 0,Y 176.353,Z 540.946,A -85,B 0,C 180,E1 -22772.288,E2 -22772.288} C_VEL
LIN {X 0,Y 176.32,Z 539.531,A -85,B 0,C 180,E1 -22775.297,E2 -22775.297} C_VEL
LIN {X 0,Y 176.617,Z 536.63,A -85,B 0,C 180,E1 -22779.163,E2 -22779.163} C_VEL
LIN {X 0,Y 177.373,Z 532.945,A -85,B 0,C 180,E1 -22782.591,E2 -22782.591} C_VEL
LIN {X 0,Y 178.063,Z 530.115,A -85,B 0,C 180,E1 -22784.691,E2 -22784.691} C_VEL
LIN {X 0,Y 178.114,Z 527.512,A -85,B 0,C 180,E1 -22786.401,E2 -22786.401} C_VEL
LIN {X 0,Y 176.72,Z 522.724,A -85,B 0,C 180,E1 -22789.176,E2 -22789.176} C_VEL
LIN {X 0,Y 175.663,Z 517.394,A -85,B 0,C 180,E1 -22791.873,E2 -22791.873} C_VEL
LIN {X 0,Y 176.236,Z 513.794,A -85,B 0,C 180,E1 -22793.408,E2 -22793.408} C_VEL
LIN {X 0,Y 178.905,Z 505.729,A -85,B 0,C 180,E1 -22796.232,E2 -22796.232} C_VEL
LIN {X 0,Y 181.082,Z 498.218,A -85,B 0,C 180,E1 -22798.392,E2 -22798.392} C_VEL
LIN {X 0,Y 181.776,Z 488.485,A -85,B 0,C 180,E1 -22800.941,E2 -22800.941} C_VEL
LIN {X 0,Y 181.777,Z 477.977,A -85,B 0,C 180,E1 -22803.301,E2 -22803.301} C_VEL
LIN {X 0,Y 181.115,Z 465.965,A -85,B 0,C 180,E1 -22805.6,E2 -22805.6} C_VEL
LIN {X 0,Y 179.853,Z 455.824,A -85,B 0,C 180,E1 -22807.315,E2 -22807.315} C_VEL
LIN {X 0,Y 177.545,Z 443.718,A -85,B 0,C 180,E1 -22809.146,E2 -22809.146} C_VEL
LIN {X 0,Y 175.325,Z 437.465,A -85,B 0,C 180,E1 -22810.17,E2 -22810.17} C_VEL
LIN {X 0,Y 174.154,Z 434.215,A -85,B 0,C 180,E1 -22810.667,E2 -22810.667} C_VEL
LIN {X 0,Y 174.107,Z 433.817,A -85,B 0,C 180,E1 -22810.729,E2 -22810.729} C_VEL
LIN {X 0,Y 173.548,Z 430.476,A -85,B 0,C 180,E1 -22814.956,E2 -22814.956} C_VEL
LIN {X 0,Y 172.68,Z 426.321,A -85,B 0,C 180,E1 -22820.656,E2 -22820.656} C_VEL
LIN {X 0,Y 172.147,Z 423.322,A -85,B 0,C 180,E1 -22825.141,E2 -22825.141} C_VEL
LIN {X 0,Y 171.62,Z 419.921,A -85,B 0,C 180,E1 -22830.566,E2 -22830.566} C_VEL
LIN {X 0,Y 171.432,Z 419.133,A -85,B 0,C 180,E1 -22832.204,E2 -22832.204} C_VEL
LIN {X 0,Y 171.463,Z 419.128,A -85,B 0,C 180,E1 -22835.802,E2 -22835.802} C_VEL
LIN {X 0,Y 171.59,Z 419.118,A -85,B 0,C 180,E1 -22840.873,E2 -22840.873} C_VEL
LIN {X 0,Y 171.585,Z 419.118,A -85,B 0,C 180,E1 -22845.773,E2 -22845.773} C_VEL
LIN {X 0,Y 171.858,Z 419.082,A -85,B 0,C 180,E1 -22850.585,E2 -22850.585} C_VEL
LIN {X 0,Y 171.823,Z 419.083,A -85,B 0,C 180,E1 -22855.307,E2 -22855.307} C_VEL
LIN {X 0,Y 172.34,Z 419.018,A -85,B 0,C 180,E1 -22860,E2 -22860} C_VEL
LIN {X 0,Y 171.828,Z 419.059,A -85,B 0,C 180,E1 -22864.692,E2 -22864.692} C_VEL
LIN {X 0,Y 171.899,Z 419.054,A -85,B 0,C 180,E1 -22869.412,E2 -22869.412} C_VEL
LIN {X 0,Y 171.619,Z 419.106,A -85,B 0,C 180,E1 -22874.223,E2 -22874.223} C_VEL
LIN {X 0,Y 171.554,Z 419.08,A -85,B 0,C 180,E1 -22879.56,E2 -22879.56} C_VEL
LIN {X 0,Y 171.472,Z 419.125,A -85,B 0,C 180,E1 -22885.61,E2 -22885.61} C_VEL
LIN {X 0,Y 171.449,Z 419.109,A -85,B 0,C 180,E1 -22890.583,E2 -22890.583} C_VEL
LIN {X 0,Y 171.401,Z 419.119,A -85,B 0,C 180,E1 -22895.033,E2 -22895.033} C_VEL
LIN {X 0,Y 171.366,Z 419.139,A -85,B 0,C 180,E1 -22898.805,E2 -22898.805} C_VEL
LIN {X 0,Y 171.332,Z 419.119,A -85,B 0,C 180,E1 -22904.213,E2 -22904.213} C_VEL
LIN {X 0,Y 171.343,Z 419.142,A -85,B 0,C 180,E1 -22908.979,E2 -22908.979} C_VEL
LIN {X 0,Y 171.394,Z 419.119,A -85,B 0,C 180,E1 -22912.038,E2 -22912.038} C_VEL
LIN {X 0,Y 171.405,Z 419.132,A -85,B 0,C 180,E1 -22915.089,E2 -22915.089} C_VEL
LIN {X 0,Y 171.456,Z 419.119,A -85,B 0,C 180,E1 -22920.531,E2 -22920.531} C_VEL
LIN {X 0,Y 171.464,Z 419.121,A -85,B 0,C 180,E1 -22925.798,E2 -22925.798} C_VEL
LIN {X 0,Y 171.612,Z 419.106,A -85,B 0,C 180,E1 -22932.031,E2 -22932.031} C_VEL
LIN {X 0,Y 172.558,Z 421.899,A -85,B 0,C 180,E1 -22932.515,E2 -22932.515} C_VEL
LIN {X 0,Y 174.028,Z 424.416,A -85,B 0,C 180,E1 -22933.098,E2 -22933.098} C_VEL
LIN {X 0,Y 178.75,Z 433.845,A -85,B 0,C 180,E1 -22935.197,E2 -22935.197} C_VEL
LIN {X 0,Y 181.86,Z 442.333,A -85,B 0,C 180,E1 -22937.02,E2 -22937.02} C_VEL
LIN {X 0,Y 183.655,Z 450.333,A -85,B 0,C 180,E1 -22938.691,E2 -22938.691} C_VEL
LIN {X 0,Y 185.385,Z 461.647,A -85,B 0,C 180,E1 -22941.274,E2 -22941.274} C_VEL
LIN {X 0,Y 186.033,Z 467.112,A -85,B 0,C 180,E1 -22942.657,E2 -22942.657} C_VEL
LIN {X 0,Y 183.452,Z 476.949,A -85,B 0,C 180,E1 -22944.908,E2 -22944.908} C_VEL
LIN {X 0,Y 180.299,Z 486.861,A -85,B 0,C 180,E1 -22947.762,E2 -22947.762} C_VEL
LIN {X 0,Y 177.227,Z 495.987,A -85,B 0,C 180,E1 -22951.132,E2 -22951.132} C_VEL
LIN {X 0,Y 174.637,Z 503.25,A -85,B 0,C 180,E1 -22954.612,E2 -22954.612} C_VEL
LIN {X 0,Y 172.627,Z 509.031,A -85,B 0,C 180,E1 -22958.187,E2 -22958.187} C_VEL
LIN {X 0,Y 171.103,Z 513.558,A -85,B 0,C 180,E1 -22961.846,E2 -22961.846} C_VEL
LIN {X 0,Y 170.276,Z 515.973,A -85,B 0,C 180,E1 -22964.333,E2 -22964.333} C_VEL
LIN {X 0,Y 169.507,Z 518.28,A -85,B 0,C 180,E1 -22967.52,E2 -22967.52} C_VEL
LIN {X 0,Y 169.085,Z 520.285,A -85,B 0,C 180,E1 -22971.962,E2 -22971.962} C_VEL
LIN {X 0,Y 169.166,Z 520.777,A -85,B 0,C 180,E1 -22974.542,E2 -22974.542} C_VEL
LIN {X 0,Y 169.448,Z 520.838,A -85,B 0,C 180,E1 -22977.139,E2 -22977.139} C_VEL
LIN {X 0,Y 170.016,Z 520.431,A -85,B 0,C 180,E1 -22979.764,E2 -22979.764} C_VEL
LIN {X 0,Y 170.767,Z 519.525,A -85,B 0,C 180,E1 -22982.339,E2 -22982.339} C_VEL
LIN {X 0,Y 171.861,Z 518.041,A -85,B 0,C 180,E1 -22985.128,E2 -22985.128} C_VEL
LIN {X 0,Y 173.769,Z 515.097,A -85,B 0,C 180,E1 -22988.814,E2 -22988.814} C_VEL
LIN {X 0,Y 176.415,Z 510.717,A -85,B 0,C 180,E1 -22992.622,E2 -22992.622} C_VEL
LIN {X 0,Y 179.697,Z 504.87,A -85,B 0,C 180,E1 -22996.34,E2 -22996.34} C_VEL
LIN {X 0,Y 182.804,Z 499.038,A -85,B 0,C 180,E1 -22999.189,E2 -22999.189} C_VEL
LIN {X 0,Y 186.654,Z 491.107,A -85,B 0,C 180,E1 -23002.243,E2 -23002.243} C_VEL
LIN {X 0,Y 190.353,Z 482.721,A -85,B 0,C 180,E1 -23004.764,E2 -23004.764} C_VEL
LIN {X 0,Y 192.596,Z 477.104,A -85,B 0,C 180,E1 -23006.152,E2 -23006.152} C_VEL
LIN {X 0,Y 192.946,Z 474.57,A -85,B 0,C 180,E1 -23006.896,E2 -23006.896} C_VEL
LIN {X 0,Y 192.277,Z 465.266,A -85,B 0,C 180,E1 -23009.829,E2 -23009.829} C_VEL
LIN {X 0,Y 190.706,Z 456.893,A -85,B 0,C 180,E1 -23012.452,E2 -23012.452} C_VEL
LIN {X 0,Y 188.143,Z 448.827,A -85,B 0,C 180,E1 -23015.15,E2 -23015.15} C_VEL
LIN {X 0,Y 184.438,Z 440.814,A -85,B 0,C 180,E1 -23018.191,E2 -23018.191} C_VEL
LIN {X 0,Y 181.213,Z 435.347,A -85,B 0,C 180,E1 -23020.581,E2 -23020.581} C_VEL
LIN {X 0,Y 179.024,Z 431.516,A -85,B 0,C 180,E1 -23022.287,E2 -23022.287} C_VEL
LIN {X 0,Y 176.695,Z 428.488,A -85,B 0,C 180,E1 -23023.982,E2 -23023.982} C_VEL
LIN {X 0,Y 175.747,Z 426.704,A -85,B 0,C 180,E1 -23024.786,E2 -23024.786} C_VEL
LIN {X 0,Y 173.274,Z 424.253,A -85,B 0,C 180,E1 -23026.606,E2 -23026.606} C_VEL
LIN {X 0,Y 172.17,Z 421.805,A -85,B 0,C 180,E1 -23027.678,E2 -23027.678} C_VEL
LIN {X 0,Y 172.087,Z 421.448,A -85,B 0,C 180,E1 -23027.906,E2 -23027.906} C_VEL
LIN {X 0,Y 172.2,Z 421.023,A -85,B 0,C 180,E1 -23030.604,E2 -23030.604} C_VEL
LIN {X 0,Y 172.096,Z 420.595,A -85,B 0,C 180,E1 -23035.315,E2 -23035.315} C_VEL
LIN {X 0,Y 172.528,Z 420.329,A -85,B 0,C 180,E1 -23040,E2 -23040} C_VEL
LIN {X 0,Y 172.119,Z 420.596,A -85,B 0,C 180,E1 -23044.684,E2 -23044.684} C_VEL
LIN {X 0,Y 172.217,Z 421.061,A -85,B 0,C 180,E1 -23049.395,E2 -23049.395} C_VEL
LIN {X 0,Y 172.132,Z 421.932,A -85,B 0,C 180,E1 -23054.181,E2 -23054.181} C_VEL
LIN {X 0,Y 172.307,Z 423.121,A -85,B 0,C 180,E1 -23059.045,E2 -23059.045} C_VEL
LIN {X 0,Y 172.525,Z 424.729,A -85,B 0,C 180,E1 -23064.039,E2 -23064.039} C_VEL
LIN {X 0,Y 172.777,Z 426.814,A -85,B 0,C 180,E1 -23069.218,E2 -23069.218} C_VEL
LIN {X 0,Y 173.229,Z 429.388,A -85,B 0,C 180,E1 -23074.61,E2 -23074.61} C_VEL
LIN {X 0,Y 173.359,Z 430.233,A -85,B 0,C 180,E1 -23075.948,E2 -23075.948} C_VEL
LIN {X 0,Y 174.507,Z 433.254,A -85,B 0,C 180,E1 -23076.983,E2 -23076.983} C_VEL
LIN {X 0,Y 177.456,Z 437.131,A -85,B 0,C 180,E1 -23079.07,E2 -23079.07} C_VEL
LIN {X 0,Y 179.15,Z 440.813,A -85,B 0,C 180,E1 -23080.43,E2 -23080.43} C_VEL
LIN {X 0,Y 180.925,Z 443.472,A -85,B 0,C 180,E1 -23081.607,E2 -23081.607} C_VEL
LIN {X 0,Y 183.124,Z 447.931,A -85,B 0,C 180,E1 -23083.231,E2 -23083.231} C_VEL
LIN {X 0,Y 187.12,Z 457.235,A -85,B 0,C 180,E1 -23086.305,E2 -23086.305} C_VEL
LIN {X 0,Y 188.452,Z 463.045,A -85,B 0,C 180,E1 -23087.841,E2 -23087.841} C_VEL
LIN {X 0,Y 189.378,Z 473.335,A -85,B 0,C 180,E1 -23090.314,E2 -23090.314} C_VEL
LIN {X 0,Y 189.268,Z 483.468,A -85,B 0,C 180,E1 -23092.786,E2 -23092.786} C_VEL
LIN {X 0,Y 188.4,Z 492.489,A -85,B 0,C 180,E1 -23095.153,E2 -23095.153} C_VEL
LIN {X 0,Y 186.801,Z 500.942,A -85,B 0,C 180,E1 -23097.585,E2 -23097.585} C_VEL
LIN {X 0,Y 185.32,Z 506.108,A -85,B 0,C 180,E1 -23099.211,E2 -23099.211} C_VEL
LIN {X 0,Y 181.161,Z 514.993,A -85,B 0,C 180,E1 -23102.261,E2 -23102.261} C_VEL
LIN {X 0,Y 177.69,Z 522.188,A -85,B 0,C 180,E1 -23105.464,E2 -23105.464} C_VEL
LIN {X 0,Y 174.819,Z 527.995,A -85,B 0,C 180,E1 -23108.794,E2 -23108.794} C_VEL
LIN {X 0,Y 172.504,Z 532.614,A -85,B 0,C 180,E1 -23112.213,E2 -23112.213} C_VEL
LIN {X 0,Y 170.76,Z 536.172,A -85,B 0,C 180,E1 -23115.708,E2 -23115.708} C_VEL
LIN {X 0,Y 170.036,Z 537.988,A -85,B 0,C 180,E1 -23118.078,E2 -23118.078} C_VEL
LIN {X 0,Y 169.237,Z 540.421,A -85,B 0,C 180,E1 -23122.848,E2 -23122.848} C_VEL
LIN {X 0,Y 169.15,Z 541.119,A -85,B 0,C 180,E1 -23125.695,E2 -23125.695} C_VEL
LIN {X 0,Y 169.409,Z 541.07,A -85,B 0,C 180,E1 -23130.005,E2 -23130.005} C_VEL
LIN {X 0,Y 169.271,Z 540.451,A -85,B 0,C 180,E1 -23132.384,E2 -23132.384} C_VEL
LIN {X 0,Y 169.259,Z 539.433,A -85,B 0,C 180,E1 -23134.768,E2 -23134.768} C_VEL
LIN {X 0,Y 169.322,Z 537.953,A -85,B 0,C 180,E1 -23137.158,E2 -23137.158} C_VEL
LIN {X 0,Y 169.816,Z 534.921,A -85,B 0,C 180,E1 -23140.738,E2 -23140.738} C_VEL
LIN {X 0,Y 171.025,Z 529.9,A -85,B 0,C 180,E1 -23144.956,E2 -23144.956} C_VEL
LIN {X 0,Y 173.123,Z 523.489,A -85,B 0,C 180,E1 -23148.956,E2 -23148.956} C_VEL
LIN {X 0,Y 175.424,Z 516.478,A -85,B 0,C 180,E1 -23152.305,E2 -23152.305} C_VEL
LIN {X 0,Y 176.236,Z 513.794,A -85,B 0,C 180,E1 -23153.408,E2 -23153.408} C_VEL
LIN {X 0,Y 176.88,Z 510.069,A -85,B 0,C 180,E1 -23154.891,E2 -23154.891} C_VEL
LIN {X 0,Y 176.604,Z 506.224,A -85,B 0,C 180,E1 -23156.368,E2 -23156.368} C_VEL
LIN {X 0,Y 175.135,Z 498.062,A -85,B 0,C 180,E1 -23159.221,E2 -23159.221} C_VEL
LIN {X 0,Y 174.919,Z 492.039,A -85,B 0,C 180,E1 -23160.962,E2 -23160.962} C_VEL
LIN {X 0,Y 175.244,Z 481.18,A -85,B 0,C 180,E1 -23163.643,E2 -23163.643} C_VEL
LIN {X 0,Y 174.921,Z 469.966,A -85,B 0,C 180,E1 -23166.017,E2 -23166.017} C_VEL
LIN {X 0,Y 173.822,Z 458.606,A -85,B 0,C 180,E1 -23168.126,E2 -23168.126} C_VEL
LIN {X 0,Y 171.754,Z 446.543,A -85,B 0,C 180,E1 -23170.122,E2 -23170.122} C_VEL
LIN {X 0,Y 169.621,Z 440.554,A -85,B 0,C 180,E1 -23171.211,E2 -23171.211} C_VEL
LIN {X 0,Y 168.237,Z 437.162,A -85,B 0,C 180,E1 -23171.829,E2 -23171.829} C_VEL
LIN {X 0,Y 166.965,Z 433.936,A -85,B 0,C 180,E1 -23172.398,E2 -23172.398} C_VEL
LIN {X 0,Y 166.842,Z 433.302,A -85,B 0,C 180,E1 -23172.526,E2 -23172.526} C_VEL
LIN {X 0,Y 166.12,Z 429.736,A -85,B 0,C 180,E1 -23177.397,E2 -23177.397} C_VEL
LIN {X 0,Y 165.702,Z 427.618,A -85,B 0,C 180,E1 -23180.49,E2 -23180.49} C_VEL
LIN {X 0,Y 165.008,Z 423.824,A -85,B 0,C 180,E1 -23186.379,E2 -23186.379} C_VEL
LIN {X 0,Y 164.808,Z 422.088,A -85,B 0,C 180,E1 -23189.221,E2 -23189.221} C_VEL
LIN {X 0,Y 164.391,Z 420.007,A -85,B 0,C 180,E1 -23193.036,E2 -23193.036} C_VEL
LIN {X 0,Y 164.388,Z 420.009,A -85,B 0,C 180,E1 -23197.37,E2 -23197.37} C_VEL
LIN {X 0,Y 164.495,Z 420,A -85,B 0,C 180,E1 -23200.052,E2 -23200.052} C_VEL
LIN {X 0,Y 164.515,Z 419.999,A -85,B 0,C 180,E1 -23205.148,E2 -23205.148} C_VEL
LIN {X 0,Y 164.779,Z 419.965,A -85,B 0,C 180,E1 -23210.177,E2 -23210.177} C_VEL
LIN {X 0,Y 164.84,Z 419.955,A -85,B 0,C 180,E1 -23212.651,E2 -23212.651} C_VEL
LIN {X 0,Y 165.056,Z 419.925,A -85,B 0,C 180,E1 -23217.559,E2 -23217.559} C_VEL
LIN {X 0,Y 165.303,Z 419.895,A -85,B 0,C 180,E1 -23220,E2 -23220} C_VEL
LIN {X 0,Y 164.778,Z 419.932,A -85,B 0,C 180,E1 -23224.893,E2 -23224.893} C_VEL
LIN {X 0,Y 164.86,Z 419.91,A -85,B 0,C 180,E1 -23227.347,E2 -23227.347} C_VEL
LIN {X 0,Y 164.764,Z 419.954,A -85,B 0,C 180,E1 -23231.15,E2 -23231.15} C_VEL
LIN {X 0,Y 164.515,Z 419.973,A -85,B 0,C 180,E1 -23237.4,E2 -23237.4} C_VEL
LIN {X 0,Y 164.484,Z 419.958,A -85,B 0,C 180,E1 -23239.988,E2 -23239.988} C_VEL
LIN {X 0,Y 164.398,Z 420.007,A -85,B 0,C 180,E1 -23246.128,E2 -23246.128} C_VEL
LIN {X 0,Y 164.383,Z 419.981,A -85,B 0,C 180,E1 -23251.225,E2 -23251.225} C_VEL
LIN {X 0,Y 164.303,Z 420.014,A -85,B 0,C 180,E1 -23256.787,E2 -23256.787} C_VEL
LIN {X 0,Y 164.299,Z 420.016,A -85,B 0,C 180,E1 -23259.914,E2 -23259.914} C_VEL
LIN {X 0,Y 164.288,Z 419.995,A -85,B 0,C 180,E1 -23263.339,E2 -23263.339} C_VEL
LIN {X 0,Y 164.3,Z 420.014,A -85,B 0,C 180,E1 -23266.806,E2 -23266.806} C_VEL
LIN {X 0,Y 164.303,Z 420.012,A -85,B 0,C 180,E1 -23270.349,E2 -23270.349} C_VEL
LIN {X 0,Y 164.337,Z 420.007,A -85,B 0,C 180,E1 -23274.346,E2 -23274.346} C_VEL
LIN {X 0,Y 164.397,Z 419.998,A -85,B 0,C 180,E1 -23279.131,E2 -23279.131} C_VEL
LIN {X 0,Y 164.422,Z 420.003,A -85,B 0,C 180,E1 -23284.69,E2 -23284.69} C_VEL
LIN {X 0,Y 164.505,Z 420.036,A -85,B 0,C 180,E1 -23290.311,E2 -23290.311} C_VEL
LIN {X 0,Y 165.533,Z 422.785,A -85,B 0,C 180,E1 -23290.83,E2 -23290.83} C_VEL
LIN {X 0,Y 166.849,Z 424.842,A -85,B 0,C 180,E1 -23291.375,E2 -23291.375} C_VEL
LIN {X 0,Y 171.825,Z 434.533,A -85,B 0,C 180,E1 -23293.725,E2 -23293.725} C_VEL
LIN {X 0,Y 175.169,Z 443.037,A -85,B 0,C 180,E1 -23295.736,E2 -23295.736} C_VEL
LIN {X 0,Y 177.092,Z 450.432,A -85,B 0,C 180,E1 -23297.417,E2 -23297.417} C_VEL
LIN {X 0,Y 178.717,Z 461.663,A -85,B 0,C 180,E1 -23300.069,E2 -23300.069} C_VEL
LIN {X 0,Y 179.438,Z 468.388,A -85,B 0,C 180,E1 -23301.843,E2 -23301.843} C_VEL
LIN {X 0,Y 177.957,Z 474.163,A -85,B 0,C 180,E1 -23303.191,E2 -23303.191} C_VEL
LIN {X 0,Y 174.726,Z 484.266,A -85,B 0,C 180,E1 -23305.959,E2 -23305.959} C_VEL
LIN {X 0,Y 171.908,Z 492.517,A -85,B 0,C 180,E1 -23308.824,E2 -23308.824} C_VEL
LIN {X 0,Y 168.906,Z 500.585,A -85,B 0,C 180,E1 -23312.38,E2 -23312.38} C_VEL
LIN {X 0,Y 166.541,Z 507.006,A -85,B 0,C 180,E1 -23316.051,E2 -23316.051} C_VEL
LIN {X 0,Y 164.723,Z 512.088,A -85,B 0,C 180,E1 -23319.821,E2 -23319.821} C_VEL
LIN {X 0,Y 163.354,Z 515.992,A -85,B 0,C 180,E1 -23323.682,E2 -23323.682} C_VEL
LIN {X 0,Y 162.361,Z 518.893,A -85,B 0,C 180,E1 -23327.769,E2 -23327.769} C_VEL
LIN {X 0,Y 162.08,Z 520.103,A -85,B 0,C 180,E1 -23330.292,E2 -23330.292} C_VEL
LIN {X 0,Y 162.073,Z 521.179,A -85,B 0,C 180,E1 -23334.408,E2 -23334.408} C_VEL
LIN {X 0,Y 162.578,Z 521.208,A -85,B 0,C 180,E1 -23338.387,E2 -23338.387} C_VEL
LIN {X 0,Y 163.262,Z 520.63,A -85,B 0,C 180,E1 -23341.096,E2 -23341.096} C_VEL
LIN {X 0,Y 164.165,Z 519.607,A -85,B 0,C 180,E1 -23343.81,E2 -23343.81} C_VEL
LIN {X 0,Y 166.022,Z 517.095,A -85,B 0,C 180,E1 -23347.859,E2 -23347.859} C_VEL
LIN {X 0,Y 168.585,Z 513.331,A -85,B 0,C 180,E1 -23351.83,E2 -23351.83} C_VEL
LIN {X 0,Y 172.039,Z 507.725,A -85,B 0,C 180,E1 -23356.015,E2 -23356.015} C_VEL
LIN {X 0,Y 175.681,Z 501.484,A -85,B 0,C 180,E1 -23359.463,E2 -23359.463} C_VEL
LIN {X 0,Y 179.375,Z 494.427,A -85,B 0,C 180,E1 -23362.496,E2 -23362.496} C_VEL
LIN {X 0,Y 183.8,Z 485.275,A -85,B 0,C 180,E1 -23365.493,E2 -23365.493} C_VEL
LIN {X 0,Y 186.775,Z 478.305,A -85,B 0,C 180,E1 -23367.343,E2 -23367.343} C_VEL
LIN {X 0,Y 186.813,Z 471.944,A -85,B 0,C 180,E1 -23369.479,E2 -23369.479} C_VEL
LIN {X 0,Y 185.836,Z 463.149,A -85,B 0,C 180,E1 -23372.439,E2 -23372.439} C_VEL
LIN {X 0,Y 183.969,Z 455.469,A -85,B 0,C 180,E1 -23375.152,E2 -23375.152} C_VEL
LIN {X 0,Y 181.404,Z 448.718,A -85,B 0,C 180,E1 -23377.807,E2 -23377.807} C_VEL
LIN {X 0,Y 178.535,Z 442.587,A -85,B 0,C 180,E1 -23380.452,E2 -23380.452} C_VEL
LIN {X 0,Y 174.657,Z 436.271,A -85,B 0,C 180,E1 -23383.734,E2 -23383.734} C_VEL
LIN {X 0,Y 172.663,Z 432.836,A -85,B 0,C 180,E1 -23385.562,E2 -23385.562} C_VEL
LIN {X 0,Y 170.21,Z 429.817,A -85,B 0,C 180,E1 -23387.708,E2 -23387.708} C_VEL
LIN {X 0,Y 169.353,Z 427.868,A -85,B 0,C 180,E1 -23388.68,E2 -23388.68} C_VEL
LIN {X 0,Y 166.63,Z 425.409,A -85,B 0,C 180,E1 -23391.206,E2 -23391.206} C_VEL
LIN {X 0,Y 165.393,Z 422.956,A -85,B 0,C 180,E1 -23392.753,E2 -23392.753} C_VEL
LIN {X 0,Y 165.263,Z 422.487,A -85,B 0,C 180,E1 -23392.977,E2 -23392.977} C_VEL
LIN {X 0,Y 165.648,Z 422.09,A -85,B 0,C 180,E1 -23400,E2 -23400} C_VEL
LIN {X 0,Y 165.246,Z 422.383,A -85,B 0,C 180,E1 -23404.88,E2 -23404.88} C_VEL
LIN {X 0,Y 165.322,Z 422.901,A -85,B 0,C 180,E1 -23409.791,E2 -23409.791} C_VEL
LIN {X 0,Y 165.259,Z 423.829,A -85,B 0,C 180,E1 -23414.783,E2 -23414.783} C_VEL
LIN {X 0,Y 165.468,Z 425.09,A -85,B 0,C 180,E1 -23419.864,E2 -23419.864} C_VEL
LIN {X 0,Y 165.656,Z 426.81,A -85,B 0,C 180,E1 -23425.104,E2 -23425.104} C_VEL
LIN {X 0,Y 166.004,Z 429.209,A -85,B 0,C 180,E1 -23430.617,E2 -23430.617} C_VEL
LIN {X 0,Y 167.462,Z 432.762,A -85,B 0,C 180,E1 -23432.333,E2 -23432.333} C_VEL
LIN {X 0,Y 170.461,Z 436.4,A -85,B 0,C 180,E1 -23434.984,E2 -23434.984} C_VEL
LIN {X 0,Y 172.107,Z 440.132,A -85,B 0,C 180,E1 -23436.627,E2 -23436.627} C_VEL
LIN {X 0,Y 174.081,Z 442.933,A -85,B 0,C 180,E1 -23438.185,E2 -23438.185} C_VEL
LIN {X 0,Y 176.042,Z 447.127,A -85,B 0,C 180,E1 -23439.947,E2 -23439.947} C_VEL
LIN {X 0,Y 177.196,Z 449.264,A -85,B 0,C 180,E1 -23440.878,E2 -23440.878} C_VEL
LIN {X 0,Y 179.233,Z 453.488,A -85,B 0,C 180,E1 -23442.577,E2 -23442.577} C_VEL
LIN {X 0,Y 182.335,Z 461.806,A -85,B 0,C 180,E1 -23445.488,E2 -23445.488} C_VEL
LIN {X 0,Y 183.337,Z 467.634,A -85,B 0,C 180,E1 -23447.115,E2 -23447.115} C_VEL
LIN {X 0,Y 183.704,Z 478.505,A -85,B 0,C 180,E1 -23449.92,E2 -23449.92} C_VEL
LIN {X 0,Y 182.932,Z 489.368,A -85,B 0,C 180,E1 -23452.84,E2 -23452.84} C_VEL
LIN {X 0,Y 181.616,Z 497.475,A -85,B 0,C 180,E1 -23455.201,E2 -23455.201} C_VEL
LIN {X 0,Y 179.223,Z 506.289,A -85,B 0,C 180,E1 -23458.042,E2 -23458.042} C_VEL
LIN {X 0,Y 174.895,Z 515.05,A -85,B 0,C 180,E1 -23461.176,E2 -23461.176} C_VEL
LIN {X 0,Y 170.936,Z 522.636,A -85,B 0,C 180,E1 -23464.76,E2 -23464.76} C_VEL
LIN {X 0,Y 168.207,Z 527.838,A -85,B 0,C 180,E1 -23467.917,E2 -23467.917} C_VEL
LIN {X 0,Y 165.716,Z 532.393,A -85,B 0,C 180,E1 -23471.459,E2 -23471.459} C_VEL
LIN {X 0,Y 163.835,Z 535.898,A -85,B 0,C 180,E1 -23475.09,E2 -23475.09} C_VEL
LIN {X 0,Y 162.474,Z 539.056,A -85,B 0,C 180,E1 -23480.041,E2 -23480.041} C_VEL
LIN {X 0,Y 162.17,Z 540.053,A -85,B 0,C 180,E1 -23482.535,E2 -23482.535} C_VEL
LIN {X 0,Y 162.076,Z 540.728,A -85,B 0,C 180,E1 -23485.819,E2 -23485.819} C_VEL
LIN {X 0,Y 162.344,Z 540.6,A -85,B 0,C 180,E1 -23490.005,E2 -23490.005} C_VEL
LIN {X 0,Y 162.163,Z 539.087,A -85,B 0,C 180,E1 -23494.58,E2 -23494.58} C_VEL
LIN {X 0,Y 162.264,Z 537.378,A -85,B 0,C 180,E1 -23497.471,E2 -23497.471} C_VEL
LIN {X 0,Y 162.804,Z 534.287,A -85,B 0,C 180,E1 -23501.206,E2 -23501.206} C_VEL
LIN {X 0,Y 163.855,Z 530.113,A -85,B 0,C 180,E1 -23504.917,E2 -23504.917} C_VEL
LIN {X 0,Y 166.02,Z 523.748,A -85,B 0,C 180,E1 -23509.156,E2 -23509.156} C_VEL
LIN {X 0,Y 168.571,Z 516.352,A -85,B 0,C 180,E1 -23512.907,E2 -23512.907} C_VEL
LIN {X 0,Y 171.405,Z 508.066,A -85,B 0,C 180,E1 -23516.158,E2 -23516.158} C_VEL
LIN {X 0,Y 174.254,Z 499.112,A -85,B 0,C 180,E1 -23518.95,E2 -23518.95} C_VEL
LIN {X 0,Y 174.919,Z 492.039,A -85,B 0,C 180,E1 -23520.962,E2 -23520.962} C_VEL
LIN {X 0,Y 174.836,Z 489.052,A -85,B 0,C 180,E1 -23521.78,E2 -23521.78} C_VEL
